ABB RobotStudio station: BARC_MRS_STEP_OPCUA_REV2.rspag

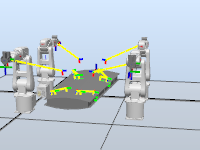
--- station ---
Station BARC_MRS_STEP_OPCUA (saved by RobotStudio 20.1.9014.1)
Controller Rob4, task T_ROB1: task frame (RAPID world) sits at (1193.8, -736.6, 0) mm, rotated rx 0 ry 0 rz -90 deg in the station
Controller Rob3, task T_ROB1: task frame (RAPID world) sits at (0, -736.6, 0) mm, rotated rx 0 ry 0 rz -90 deg in the station
Controller Rob2, task T_ROB1: task frame (RAPID world) sits at (1193.8, 0, 0) mm, rotated rx 0 ry 0 rz 90 deg in the station
Controller Rob1, task T_ROB1: task frame (RAPID world) sits at (0, 0, 0) mm, rotated rx 0 ry 0 rz 90 deg in the station
Controller Rob1
  mechanical unit ROB_1: Rob1, 6 joints, base frame (0, 0, 0) mm
Controller Rob2
  mechanical unit ROB_1: Rob2, 6 joints, base frame (0, 0, 0) mm
Controller Rob3
  mechanical unit ROB_1: Rob3, 6 joints, base frame (0, 0, 0) mm
Controller Rob4
  mechanical unit ROB_1: Rob4, 6 joints, base frame (0, 0, 0) mm
Layout (positions relative to the parent item):
  - Rob1 [mechanism, from Robots\IRB120_3_58_G_01.rslib] at (0, 0, 0) mm, rotated rx 0 ry 0 rz 90 deg; joint values [0, 0, 0, 0, 0, 0] (rad or m)
  - Rob2 [mechanism, from Robots\IRB120_3_58_G_01.rslib] at (1193.8, 0, 0) mm, rotated rx 0 ry 0 rz 90 deg; joint values [0, 0, 0, 0, 0, 0] (rad or m)
  - Rob3 [mechanism, from Robots\IRB120_3_58_G_01.rslib] at (0, -736.6, 0) mm, rotated rx 0 ry 0 rz -90 deg; joint values [0, 0, 0, 0, 0, 0] (rad or m)
  - Rob4 [mechanism, from Robots\IRB120_3_58_G_01.rslib] at (1193.8, -736.6, 0) mm, rotated rx 0 ry 0 rz -90 deg; joint values [0, 0, 0, 0, 0, 0] (rad or m)
  - MyTool [mechanism, from Training Objects\myTool.rslib] at (0, 374, 630) mm, rotated rx 0 ry 90 rz 90 deg
  - MyTool_2 [mechanism, from Training Objects\myTool.rslib] at (1193.8, 374, 630) mm, rotated rx 0 ry 90 rz 90 deg
  - MyTool_3 [mechanism, from Training Objects\myTool.rslib] at (0, -1110.6, 630) mm, rotated rx 0 ry 90 rz -90 deg
  - MyTool_4 [mechanism, from Training Objects\myTool.rslib] at (1193.8, -1110.6, 630) mm, rotated rx 0 ry 90 rz -90 deg
  - ScaledWing_Simple_Corrected [part] at (871.22, 154, 150.3) mm, rotated rx 90 ry 0 rz -90 deg
  - onepiece [part] at (287.65, 225, -913.8) mm, rotated rx 89 ry 0 rz 0 deg
  - PendEff [mechanism, from Libraries\PendEff.rslib] at (0, 374, 630) mm, rotated rx 0 ry 90 rz 90 deg
  - PendEff_2 [mechanism, from Libraries\PendEff.rslib] at (1193.8, 374, 630) mm, rotated rx 0 ry 90 rz 90 deg
  - PendEff_3 [mechanism, from Libraries\PendEff.rslib] at (0, -1110.6, 630) mm, rotated rx 0 ry 90 rz -90 deg
  - PendEff_4 [mechanism, from Libraries\PendEff.rslib] at (1193.8, -1110.6, 630) mm, rotated rx 0 ry 90 rz -90 deg
  - wing_with_holes_2 [part] at (596.5, 225, -913.8) mm, rotated rx 89 ry 0 rz 0 deg
  - Part_1 [part]
  - Part_2 [part]
  - Part_3 [part]
  - Part_4 [part]
  - Part_5 [part]
  - Part_6 [part]
  - Part_7 [part]
  - Part_8 [part]
  - partwithpoints [part, from Libraries\partwithpoints.rslib]
  - SmartComponent_1 [smart component]
Attachment: MyTool is attached to Rob1 / Link6
Attachment: MyTool_2 is attached to Rob2 / Link6
Attachment: MyTool_3 is attached to Rob3 / Link6
Attachment: MyTool_4 is attached to Rob4 / Link6
Attachment: PendEff is attached to Rob1 / Link6
Attachment: PendEff_2 is attached to Rob2 / Link6
Attachment: PendEff_3 is attached to Rob3 / Link6
Attachment: PendEff_4 is attached to Rob4 / Link6
Targets, tools, work objects and paths stored in the station and not in the controller backup, written as RAPID:
! task T_ROB1
MODULE KegleyMod
  PERS speeddata ExternalFedSpeedData:=[100,100,500,500];
  PERS zonedata ExternalFedZoneData:=[True,0,0,0,0,0,0];
ENDMODULE

! task T_ROB1
MODULE StanModule
  PROC STEPpath()
    MoveL current_robtarget,v1000,z100,PendEff_point\WObj:=A;
    SetDO doIsComplete,1;
  ENDPROC
  PROC WorkingStep()
    SetDO doIsComplete,0;
    MoveL current_robtarget,v1000,z100,PendEff_point\WObj:=A;
    SetDO doIsComplete,1;
  ENDPROC
ENDMODULE

! task T_ROB1
MODULE Targets
  CONST robtarget Drilling0:=[[255.049346094,-251.794133959,27.074601391],[0.009317717,-0.000993284,-0.994322357,-0.105996434],[0,0,0,0],[9E+09,9E+09,9E+09,9E+09,9E+09,9E+09]];
  CONST robtarget Drilling1:=[[254.118737842,-241.085099842,-22.575076921],[0.009317717,-0.000993284,-0.994322357,-0.105996434],[0,0,0,0],[9E+09,9E+09,9E+09,9E+09,9E+09,9E+09]];
  CONST robtarget Drilling2:=[[254.118737842,-241.085099842,-22.575076921],[0.009317717,-0.000993284,-0.994322357,-0.105996434],[0,0,0,0],[9E+09,9E+09,9E+09,9E+09,9E+09,9E+09]];
  CONST robtarget Drilling3:=[[253.537107684,-234.391953519,-53.606125867],[0.009317717,-0.000993284,-0.994322357,-0.105996434],[0,0,0,0],[9E+09,9E+09,9E+09,9E+09,9E+09,9E+09]];
  CONST robtarget Drilling4:=[[253.537107684,-234.391953519,-53.606125867],[0.009317717,-0.000993284,-0.994322357,-0.105996434],[0,0,0,0],[9E+09,9E+09,9E+09,9E+09,9E+09,9E+09]];
  CONST robtarget Drilling5:=[[254.118737842,-241.085099842,-22.575076921],[0.009317717,-0.000993284,-0.994322357,-0.105996434],[0,0,0,0],[9E+09,9E+09,9E+09,9E+09,9E+09,9E+09]];
  CONST robtarget Drilling6:=[[255.049346094,-251.794133959,27.074601391],[0.009317717,-0.000993284,-0.994322357,-0.105996434],[0,0,0,0],[9E+09,9E+09,9E+09,9E+09,9E+09,9E+09]];
  CONST robtarget Drilling7:=[[593.951420596,-86.046366407,46.267647759],[0.006736064,-0.000262673,-0.999217855,-0.038964529],[0,0,0,0],[9E+09,9E+09,9E+09,9E+09,9E+09,9E+09]];
  CONST robtarget Drilling8:=[[593.268611665,-82.090486811,-4.373489556],[0.006736064,-0.000262673,-0.999217855,-0.038964529],[0,0,0,0],[9E+09,9E+09,9E+09,9E+09,9E+09,9E+09]];
  CONST robtarget Drilling9:=[[593.268611665,-82.090486811,-4.373489556],[0.006736064,-0.000262673,-0.999217855,-0.038964529],[0,0,0,0],[9E+09,9E+09,9E+09,9E+09,9E+09,9E+09]];
  CONST robtarget Drilling10:=[[592.841856083,-79.618062064,-36.024200378],[0.006736064,-0.000262673,-0.999217855,-0.038964529],[0,0,0,0],[9E+09,9E+09,9E+09,9E+09,9E+09,9E+09]];
  CONST robtarget Drilling11:=[[592.841856083,-79.618062064,-36.024200378],[0.006736064,-0.000262673,-0.999217855,-0.038964529],[0,0,0,0],[9E+09,9E+09,9E+09,9E+09,9E+09,9E+09]];
  CONST robtarget Drilling12:=[[593.268611665,-82.090486811,-4.373489556],[0.006736064,-0.000262673,-0.999217855,-0.038964529],[0,0,0,0],[9E+09,9E+09,9E+09,9E+09,9E+09,9E+09]];
  CONST robtarget Drilling13:=[[593.951420596,-86.046366407,46.267647759],[0.006736064,-0.000262673,-0.999217855,-0.038964529],[0,0,0,0],[9E+09,9E+09,9E+09,9E+09,9E+09,9E+09]];
  CONST robtarget Drilling14:=[[594.013579836,-136.119059315,41.206016458],[0.007335405,-0.000453474,-0.998067656,-0.061700413],[0,0,0,0],[9E+09,9E+09,9E+09,9E+09,9E+09,9E+09]];
  CONST robtarget Drilling15:=[[593.272585499,-129.86207284,-9.201731435],[0.007335405,-0.000453474,-0.998067656,-0.061700413],[0,0,0,0],[9E+09,9E+09,9E+09,9E+09,9E+09,9E+09]];
  CONST robtarget Drilling16:=[[593.272585499,-129.86207284,-9.201731435],[0.007335405,-0.000453474,-0.998067656,-0.061700413],[0,0,0,0],[9E+09,9E+09,9E+09,9E+09,9E+09,9E+09]];
  CONST robtarget Drilling17:=[[592.809464038,-125.951456293,-40.706573868],[0.007335405,-0.000453474,-0.998067656,-0.061700413],[0,0,0,0],[9E+09,9E+09,9E+09,9E+09,9E+09,9E+09]];
  CONST robtarget Drilling18:=[[592.809464038,-125.951456293,-40.706573868],[0.007335405,-0.000453474,-0.998067656,-0.061700413],[0,0,0,0],[9E+09,9E+09,9E+09,9E+09,9E+09,9E+09]];
  CONST robtarget Drilling19:=[[593.272585499,-129.86207284,-9.201731435],[0.007335405,-0.000453474,-0.998067656,-0.061700413],[0,0,0,0],[9E+09,9E+09,9E+09,9E+09,9E+09,9E+09]];
  CONST robtarget Drilling20:=[[594.013579836,-136.119059315,41.206016458],[0.007335405,-0.000453474,-0.998067656,-0.061700413],[0,0,0,0],[9E+09,9E+09,9E+09,9E+09,9E+09,9E+09]];
  PROC dummy()
    MoveL Drilling0,v0,z10,DrillTool\WObj:=A;
    MoveL Drilling1,v1,z10,DrillTool\WObj:=A;
    MoveL Drilling2,v2,z10,DrillTool\WObj:=A;
    MoveL Drilling3,v3,z10,DrillTool\WObj:=A;
    MoveL Drilling4,v4,z10,DrillTool\WObj:=A;
    MoveL Drilling5,v5,z10,DrillTool\WObj:=A;
    MoveL Drilling6,v6,z10,DrillTool\WObj:=A;
    MoveL Drilling7,v7,z10,DrillTool\WObj:=A;
    MoveL Drilling8,v8,z10,DrillTool\WObj:=A;
    MoveL Drilling9,v9,z10,DrillTool\WObj:=A;
    MoveL Drilling10,v10,z10,DrillTool\WObj:=A;
    MoveL Drilling11,v11,z10,DrillTool\WObj:=A;
    MoveL Drilling12,v12,z10,DrillTool\WObj:=A;
    MoveL Drilling13,v13,z10,DrillTool\WObj:=A;
    MoveL Drilling14,v14,z10,DrillTool\WObj:=A;
    MoveL Drilling15,v15,z10,DrillTool\WObj:=A;
    MoveL Drilling16,v16,z10,DrillTool\WObj:=A;
    MoveL Drilling17,v17,z10,DrillTool\WObj:=A;
    MoveL Drilling18,v18,z10,DrillTool\WObj:=A;
    MoveL Drilling19,v19,z10,DrillTool\WObj:=A;
    MoveL Drilling20,v20,z10,DrillTool\WObj:=A;
  ENDPROC
ENDMODULE

! task T_ROB1
MODULE KegleyMod
  PERS speeddata ExternalFedSpeedData:=[100,100,500,500];
  PERS zonedata ExternalFedZoneData:=[True,0,0,0,0,0,0];
ENDMODULE

! task T_ROB1
MODULE KyleModule
  PROC WorkingStep()
    SetDO doIsComplete,0;
    MoveL current_robtarget,v1000,z100,PendEff_point\WObj:=A;
    SetDO doIsComplete,1;
  ENDPROC
ENDMODULE

! task T_ROB1
MODULE Targets
  CONST robtarget Drilling0:=[[241.166080887,78.477337456,51.523766918],[0.006620989,0.000217104,-0.999440903,0.032771904],[0,0,0,0],[9E+09,9E+09,9E+09,9E+09,9E+09,9E+09]];
  CONST robtarget Drilling1:=[[240.494487367,75.149427584,0.837338971],[0.006620989,0.000217104,-0.999440903,0.032771904],[0,0,0,0],[9E+09,9E+09,9E+09,9E+09,9E+09,9E+09]];
  CONST robtarget Drilling2:=[[240.494487367,75.149427584,0.837338971],[0.006620989,0.000217104,-0.999440903,0.032771904],[0,0,0,0],[9E+09,9E+09,9E+09,9E+09,9E+09,9E+09]];
  CONST robtarget Drilling3:=[[240.074741417,73.069483914,-30.841678495],[0.006620989,0.000217104,-0.999440903,0.032771904],[0,0,0,0],[9E+09,9E+09,9E+09,9E+09,9E+09,9E+09]];
  CONST robtarget Drilling4:=[[240.074741417,73.069483914,-30.841678495],[0.006620989,0.000217104,-0.999440903,0.032771904],[0,0,0,0],[9E+09,9E+09,9E+09,9E+09,9E+09,9E+09]];
  CONST robtarget Drilling5:=[[240.494487367,75.149427584,0.837338971],[0.006620989,0.000217104,-0.999440903,0.032771904],[0,0,0,0],[9E+09,9E+09,9E+09,9E+09,9E+09,9E+09]];
  CONST robtarget Drilling6:=[[241.166080887,78.477337456,51.523766918],[0.006620989,0.000217104,-0.999440903,0.032771904],[0,0,0,0],[9E+09,9E+09,9E+09,9E+09,9E+09,9E+09]];
  CONST robtarget Drilling7:=[[590.794286308,244.057268889,22.395212352],[0.009603198,0.001072712,-0.993772536,0.111007991],[0,0,0,0],[9E+09,9E+09,9E+09,9E+09,9E+09,9E+09]];
  CONST robtarget Drilling8:=[[589.836775887,232.848046285,-27.143424109],[0.009603198,0.001072712,-0.993772536,0.111007991],[0,0,0,0],[9E+09,9E+09,9E+09,9E+09,9E+09,9E+09]];
  CONST robtarget Drilling9:=[[589.836775887,232.848046285,-27.143424109],[0.009603198,0.001072712,-0.993772536,0.111007991],[0,0,0,0],[9E+09,9E+09,9E+09,9E+09,9E+09,9E+09]];
  CONST robtarget Drilling10:=[[589.238331874,225.842282157,-58.105071897],[0.009603198,0.001072712,-0.993772536,0.111007991],[0,0,0,0],[9E+09,9E+09,9E+09,9E+09,9E+09,9E+09]];
  CONST robtarget Drilling11:=[[589.238331874,225.842282157,-58.105071897],[0.009603198,0.001072712,-0.993772536,0.111007991],[0,0,0,0],[9E+09,9E+09,9E+09,9E+09,9E+09,9E+09]];
  CONST robtarget Drilling12:=[[589.836775887,232.848046285,-27.143424109],[0.009603198,0.001072712,-0.993772536,0.111007991],[0,0,0,0],[9E+09,9E+09,9E+09,9E+09,9E+09,9E+09]];
  CONST robtarget Drilling13:=[[590.794286308,244.057268889,22.395212352],[0.009603198,0.001072712,-0.993772536,0.111007991],[0,0,0,0],[9E+09,9E+09,9E+09,9E+09,9E+09,9E+09]];
  CONST robtarget Drilling14:=[[586.927237976,164.129102175,37.475265565],[0.00778853,0.000580627,-0.997202343,0.074340359],[0,0,0,0],[9E+09,9E+09,9E+09,9E+09,9E+09,9E+09]];
  CONST robtarget Drilling15:=[[586.142522602,156.59679287,-12.757079974],[0.00778853,0.000580627,-0.997202343,0.074340359],[0,0,0,0],[9E+09,9E+09,9E+09,9E+09,9E+09,9E+09]];
  CONST robtarget Drilling16:=[[586.142522602,156.59679287,-12.757079974],[0.00778853,0.000580627,-0.997202343,0.074340359],[0,0,0,0],[9E+09,9E+09,9E+09,9E+09,9E+09,9E+09]];
  CONST robtarget Drilling17:=[[585.652075493,151.889099555,-44.152295936],[0.00778853,0.000580627,-0.997202343,0.074340359],[0,0,0,0],[9E+09,9E+09,9E+09,9E+09,9E+09,9E+09]];
  CONST robtarget Drilling18:=[[585.652075493,151.889099555,-44.152295936],[0.00778853,0.000580627,-0.997202343,0.074340359],[0,0,0,0],[9E+09,9E+09,9E+09,9E+09,9E+09,9E+09]];
  CONST robtarget Drilling19:=[[586.142522602,156.59679287,-12.757079974],[0.00778853,0.000580627,-0.997202343,0.074340359],[0,0,0,0],[9E+09,9E+09,9E+09,9E+09,9E+09,9E+09]];
  CONST robtarget Drilling20:=[[586.927237976,164.129102175,37.475265565],[0.00778853,0.000580627,-0.997202343,0.074340359],[0,0,0,0],[9E+09,9E+09,9E+09,9E+09,9E+09,9E+09]];
  PROC dummy()
    MoveL Drilling0,v0,z10,DrillTool\WObj:=A;
    MoveL Drilling1,v1,z10,DrillTool\WObj:=A;
    MoveL Drilling2,v2,z10,DrillTool\WObj:=A;
    MoveL Drilling3,v3,z10,DrillTool\WObj:=A;
    MoveL Drilling4,v4,z10,DrillTool\WObj:=A;
    MoveL Drilling5,v5,z10,DrillTool\WObj:=A;
    MoveL Drilling6,v6,z10,DrillTool\WObj:=A;
    MoveL Drilling7,v7,z10,DrillTool\WObj:=A;
    MoveL Drilling8,v8,z10,DrillTool\WObj:=A;
    MoveL Drilling9,v9,z10,DrillTool\WObj:=A;
    MoveL Drilling10,v10,z10,DrillTool\WObj:=A;
    MoveL Drilling11,v11,z10,DrillTool\WObj:=A;
    MoveL Drilling12,v12,z10,DrillTool\WObj:=A;
    MoveL Drilling13,v13,z10,DrillTool\WObj:=A;
    MoveL Drilling14,v14,z10,DrillTool\WObj:=A;
    MoveL Drilling15,v15,z10,DrillTool\WObj:=A;
    MoveL Drilling16,v16,z10,DrillTool\WObj:=A;
    MoveL Drilling17,v17,z10,DrillTool\WObj:=A;
    MoveL Drilling18,v18,z10,DrillTool\WObj:=A;
    MoveL Drilling19,v19,z10,DrillTool\WObj:=A;
    MoveL Drilling20,v20,z10,DrillTool\WObj:=A;
  ENDPROC
ENDMODULE

! task T_ROB1
MODULE KegleyMod
  PERS speeddata ExternalFedSpeedData:=[100,100,500,500];
  PERS zonedata ExternalFedZoneData:=[True,0,0,0,0,0,0];
ENDMODULE

! task T_ROB1
MODULE CartmanWorkingPlan
  PROC WorkingStep()
    SetDO doIsComplete,0;
    MoveL current_robtarget,v1000,z100,PendEff_point\WObj:=A;
    SetDO doIsComplete,1;
  ENDPROC
ENDMODULE

! task T_ROB1
MODULE Targets
  CONST robtarget Drilling0:=[[1189.808543498,-65.923675679,39.773088683],[0.006653359,-0.000231419,-0.9993735,-0.034760413],[0,0,0,0],[9E+09,9E+09,9E+09,9E+09,9E+09,9E+09]];
  CONST robtarget Drilling1:=[[1189.133802971,-62.394073863,-10.899651881],[0.006653359,-0.000231419,-0.9993735,-0.034760413],[0,0,0,0],[9E+09,9E+09,9E+09,9E+09,9E+09,9E+09]];
  CONST robtarget Drilling2:=[[1189.133802971,-62.394073863,-10.899651881],[0.006653359,-0.000231419,-0.9993735,-0.034760413],[0,0,0,0],[9E+09,9E+09,9E+09,9E+09,9E+09,9E+09]];
  CONST robtarget Drilling3:=[[1188.712090141,-60.188072728,-42.570114734],[0.006653359,-0.000231419,-0.9993735,-0.034760413],[0,0,0,0],[9E+09,9E+09,9E+09,9E+09,9E+09,9E+09]];
  CONST robtarget Drilling4:=[[1188.712090141,-60.188072728,-42.570114734],[0.006653359,-0.000231419,-0.9993735,-0.034760413],[0,0,0,0],[9E+09,9E+09,9E+09,9E+09,9E+09,9E+09]];
  CONST robtarget Drilling5:=[[1189.133802971,-62.394073863,-10.899651881],[0.006653359,-0.000231419,-0.9993735,-0.034760413],[0,0,0,0],[9E+09,9E+09,9E+09,9E+09,9E+09,9E+09]];
  CONST robtarget Drilling6:=[[1189.808543498,-65.923675679,39.773088683],[0.006653359,-0.000231419,-0.9993735,-0.034760413],[0,0,0,0],[9E+09,9E+09,9E+09,9E+09,9E+09,9E+09]];
  CONST robtarget Drilling7:=[[1275.333810152,-199.568058709,19.231409467],[0.009422515,-0.001026722,-0.994071031,-0.10831873],[0,0,0,0],[9E+09,9E+09,9E+09,9E+09,9E+09,9E+09]];
  CONST robtarget Drilling8:=[[1274.39345782,-188.627142215,-30.367502656],[0.009422515,-0.001026722,-0.994071031,-0.10831873],[0,0,0,0],[9E+09,9E+09,9E+09,9E+09,9E+09,9E+09]];
  CONST robtarget Drilling9:=[[1274.39345782,-188.627142215,-30.367502656],[0.009422515,-0.001026722,-0.994071031,-0.10831873],[0,0,0,0],[9E+09,9E+09,9E+09,9E+09,9E+09,9E+09]];
  CONST robtarget Drilling10:=[[1273.805737613,-181.789069407,-61.366822732],[0.009422515,-0.001026722,-0.994071031,-0.10831873],[0,0,0,0],[9E+09,9E+09,9E+09,9E+09,9E+09,9E+09]];
  CONST robtarget Drilling11:=[[1273.805737613,-181.789069407,-61.366822732],[0.009422515,-0.001026722,-0.994071031,-0.10831873],[0,0,0,0],[9E+09,9E+09,9E+09,9E+09,9E+09,9E+09]];
  CONST robtarget Drilling12:=[[1274.39345782,-188.627142215,-30.367502656],[0.009422515,-0.001026722,-0.994071031,-0.10831873],[0,0,0,0],[9E+09,9E+09,9E+09,9E+09,9E+09,9E+09]];
  CONST robtarget Drilling13:=[[1275.333810152,-199.568058709,19.231409467],[0.009422515,-0.001026722,-0.994071031,-0.10831873],[0,0,0,0],[9E+09,9E+09,9E+09,9E+09,9E+09,9E+09]];
  CONST robtarget Drilling14:=[[1277.649426378,-158.123953639,27.348886106],[0.008256342,-0.000710159,-0.996287003,-0.085694437],[0,0,0,0],[9E+09,9E+09,9E+09,9E+09,9E+09,9E+09]];
  CONST robtarget Drilling15:=[[1276.819879727,-149.449130571,-22.698084803],[0.008256342,-0.000710159,-0.996287003,-0.085694437],[0,0,0,0],[9E+09,9E+09,9E+09,9E+09,9E+09,9E+09]];
  CONST robtarget Drilling16:=[[1276.819879727,-149.449130571,-22.698084803],[0.008256342,-0.000710159,-0.996287003,-0.085694437],[0,0,0,0],[9E+09,9E+09,9E+09,9E+09,9E+09,9E+09]];
  CONST robtarget Drilling17:=[[1276.30141307,-144.027366153,-53.97744162],[0.008256342,-0.000710159,-0.996287003,-0.085694437],[0,0,0,0],[9E+09,9E+09,9E+09,9E+09,9E+09,9E+09]];
  CONST robtarget Drilling18:=[[1276.30141307,-144.027366153,-53.97744162],[0.008256342,-0.000710159,-0.996287003,-0.085694437],[0,0,0,0],[9E+09,9E+09,9E+09,9E+09,9E+09,9E+09]];
  CONST robtarget Drilling19:=[[1276.819879727,-149.449130571,-22.698084803],[0.008256342,-0.000710159,-0.996287003,-0.085694437],[0,0,0,0],[9E+09,9E+09,9E+09,9E+09,9E+09,9E+09]];
  CONST robtarget Drilling20:=[[1277.649426378,-158.123953639,27.348886106],[0.008256342,-0.000710159,-0.996287003,-0.085694437],[0,0,0,0],[9E+09,9E+09,9E+09,9E+09,9E+09,9E+09]];
  PROC dummy()
    MoveL Drilling0,v0,z10,DrillTool\WObj:=A;
    MoveL Drilling1,v1,z10,DrillTool\WObj:=A;
    MoveL Drilling2,v2,z10,DrillTool\WObj:=A;
    MoveL Drilling3,v3,z10,DrillTool\WObj:=A;
    MoveL Drilling4,v4,z10,DrillTool\WObj:=A;
    MoveL Drilling5,v5,z10,DrillTool\WObj:=A;
    MoveL Drilling6,v6,z10,DrillTool\WObj:=A;
    MoveL Drilling7,v7,z10,DrillTool\WObj:=A;
    MoveL Drilling8,v8,z10,DrillTool\WObj:=A;
    MoveL Drilling9,v9,z10,DrillTool\WObj:=A;
    MoveL Drilling10,v10,z10,DrillTool\WObj:=A;
    MoveL Drilling11,v11,z10,DrillTool\WObj:=A;
    MoveL Drilling12,v12,z10,DrillTool\WObj:=A;
    MoveL Drilling13,v13,z10,DrillTool\WObj:=A;
    MoveL Drilling14,v14,z10,DrillTool\WObj:=A;
    MoveL Drilling15,v15,z10,DrillTool\WObj:=A;
    MoveL Drilling16,v16,z10,DrillTool\WObj:=A;
    MoveL Drilling17,v17,z10,DrillTool\WObj:=A;
    MoveL Drilling18,v18,z10,DrillTool\WObj:=A;
    MoveL Drilling19,v19,z10,DrillTool\WObj:=A;
    MoveL Drilling20,v20,z10,DrillTool\WObj:=A;
  ENDPROC
ENDMODULE

! task T_ROB1
MODULE KegleyMod
  PERS speeddata ExternalFedSpeedData:=[100,100,500,500];
  PERS zonedata ExternalFedZoneData:=[True,0,0,0,0,0,0];
ENDMODULE

! task T_ROB1
MODULE Targets
  CONST robtarget Drilling0:=[[1191.894155606,213.973804454,17.582383099],[0.009735859,0.001112565,-0.993486175,0.11353059],[0,0,0,0],[9E+09,9E+09,9E+09,9E+09,9E+09,9E+09]];
  CONST robtarget Drilling1:=[[1190.924268649,202.513131068,-31.898444348],[0.009735859,0.001112565,-0.993486175,0.11353059],[0,0,0,0],[9E+09,9E+09,9E+09,9E+09,9E+09,9E+09]];
  CONST robtarget Drilling2:=[[1190.924268649,202.513131068,-31.898444348],[0.009735859,0.001112565,-0.993486175,0.11353059],[0,0,0,0],[9E+09,9E+09,9E+09,9E+09,9E+09,9E+09]];
  CONST robtarget Drilling3:=[[1190.318089301,195.350210202,-62.823961503],[0.009735859,0.001112565,-0.993486175,0.11353059],[0,0,0,0],[9E+09,9E+09,9E+09,9E+09,9E+09,9E+09]];
  CONST robtarget Drilling4:=[[1190.318089301,195.350210202,-62.823961503],[0.009735859,0.001112565,-0.993486175,0.11353059],[0,0,0,0],[9E+09,9E+09,9E+09,9E+09,9E+09,9E+09]];
  CONST robtarget Drilling5:=[[1190.924268649,202.513131068,-31.898444348],[0.009735859,0.001112565,-0.993486175,0.11353059],[0,0,0,0],[9E+09,9E+09,9E+09,9E+09,9E+09,9E+09]];
  CONST robtarget Drilling6:=[[1191.894155606,213.973804454,17.582383099],[0.009735859,0.001112565,-0.993486175,0.11353059],[0,0,0,0],[9E+09,9E+09,9E+09,9E+09,9E+09,9E+09]];
  CONST robtarget Drilling7:=[[1279.805555756,62.025883801,38.843455502],[0.006631324,0.000222501,-0.999415571,0.033533444],[0,0,0,0],[9E+09,9E+09,9E+09,9E+09,9E+09,9E+09]];
  CONST robtarget Drilling8:=[[1279.132965076,58.620727156,-11.837828321],[0.006631324,0.000222501,-0.999415571,0.033533444],[0,0,0,0],[9E+09,9E+09,9E+09,9E+09,9E+09,9E+09]];
  CONST robtarget Drilling9:=[[1279.132965076,58.620727156,-11.837828321],[0.006631324,0.000222501,-0.999415571,0.033533444],[0,0,0,0],[9E+09,9E+09,9E+09,9E+09,9E+09,9E+09]];
  CONST robtarget Drilling10:=[[1278.712595901,56.492504252,-43.513630711],[0.006631324,0.000222501,-0.999415571,0.033533444],[0,0,0,0],[9E+09,9E+09,9E+09,9E+09,9E+09,9E+09]];
  CONST robtarget Drilling11:=[[1278.712595901,56.492504252,-43.513630711],[0.006631324,0.000222501,-0.999415571,0.033533444],[0,0,0,0],[9E+09,9E+09,9E+09,9E+09,9E+09,9E+09]];
  CONST robtarget Drilling12:=[[1279.132965076,58.620727156,-11.837828321],[0.006631324,0.000222501,-0.999415571,0.033533444],[0,0,0,0],[9E+09,9E+09,9E+09,9E+09,9E+09,9E+09]];
  CONST robtarget Drilling13:=[[1279.805555756,62.025883801,38.843455502],[0.006631324,0.000222501,-0.999415571,0.033533444],[0,0,0,0],[9E+09,9E+09,9E+09,9E+09,9E+09,9E+09]];
  CONST robtarget Drilling14:=[[1280.462702991,102.383093395,35.233257482],[0.007136454,0.000396072,-0.998437928,0.055413159],[0,0,0,0],[9E+09,9E+09,9E+09,9E+09,9E+09,9E+09]];
  CONST robtarget Drilling15:=[[1279.741001712,96.761623708,-15.249593327],[0.007136454,0.000396072,-0.998437928,0.055413159],[0,0,0,0],[9E+09,9E+09,9E+09,9E+09,9E+09,9E+09]];
  CONST robtarget Drilling16:=[[1279.741001712,96.761623708,-15.249593327],[0.007136454,0.000396072,-0.998437928,0.055413159],[0,0,0,0],[9E+09,9E+09,9E+09,9E+09,9E+09,9E+09]];
  CONST robtarget Drilling17:=[[1279.289938413,93.248205154,-46.801375083],[0.007136454,0.000396072,-0.998437928,0.055413159],[0,0,0,0],[9E+09,9E+09,9E+09,9E+09,9E+09,9E+09]];
  CONST robtarget Drilling18:=[[1279.289938413,93.248205154,-46.801375083],[0.007136454,0.000396072,-0.998437928,0.055413159],[0,0,0,0],[9E+09,9E+09,9E+09,9E+09,9E+09,9E+09]];
  CONST robtarget Drilling19:=[[1279.741001712,96.761623708,-15.249593327],[0.007136454,0.000396072,-0.998437928,0.055413159],[0,0,0,0],[9E+09,9E+09,9E+09,9E+09,9E+09,9E+09]];
  CONST robtarget Drilling20:=[[1280.462702991,102.383093395,35.233257482],[0.007136454,0.000396072,-0.998437928,0.055413159],[0,0,0,0],[9E+09,9E+09,9E+09,9E+09,9E+09,9E+09]];
  PROC dummy()
    MoveL Drilling0,v0,z10,DrillTool\WObj:=A;
    MoveL Drilling1,v1,z10,DrillTool\WObj:=A;
    MoveL Drilling2,v2,z10,DrillTool\WObj:=A;
    MoveL Drilling3,v3,z10,DrillTool\WObj:=A;
    MoveL Drilling4,v4,z10,DrillTool\WObj:=A;
    MoveL Drilling5,v5,z10,DrillTool\WObj:=A;
    MoveL Drilling6,v6,z10,DrillTool\WObj:=A;
    MoveL Drilling7,v7,z10,DrillTool\WObj:=A;
    MoveL Drilling8,v8,z10,DrillTool\WObj:=A;
    MoveL Drilling9,v9,z10,DrillTool\WObj:=A;
    MoveL Drilling10,v10,z10,DrillTool\WObj:=A;
    MoveL Drilling11,v11,z10,DrillTool\WObj:=A;
    MoveL Drilling12,v12,z10,DrillTool\WObj:=A;
    MoveL Drilling13,v13,z10,DrillTool\WObj:=A;
    MoveL Drilling14,v14,z10,DrillTool\WObj:=A;
    MoveL Drilling15,v15,z10,DrillTool\WObj:=A;
    MoveL Drilling16,v16,z10,DrillTool\WObj:=A;
    MoveL Drilling17,v17,z10,DrillTool\WObj:=A;
    MoveL Drilling18,v18,z10,DrillTool\WObj:=A;
    MoveL Drilling19,v19,z10,DrillTool\WObj:=A;
    MoveL Drilling20,v20,z10,DrillTool\WObj:=A;
  ENDPROC
ENDMODULE

! task T_ROB1
MODULE KennyWorkingPlan
  PROC WorkingStep()
    SetDO doIsComplete,0;
    MoveL current_robtarget,v1000,z100,PendEff_point\WObj:=A;
    SetDO doIsComplete,1;
  ENDPROC
ENDMODULE


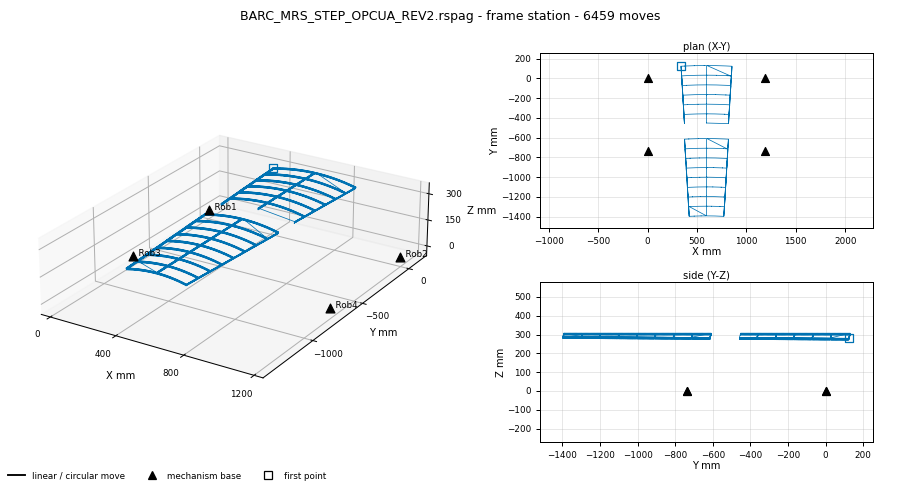
[picture p0: tool path of BARC_MRS_STEP_OPCUA_REV2.rspag in frame station, 6459 of 6483 moves have a stored position in this frame; points joined in program order, loops and branches not executed]
--- Backups/Rob1/RAPID/TASK1/PROGMOD/StanTargets.mod ---
MODULE StanTargets

	!Workplan Variables
	CONST string workplanName := "Stan";
	CONST string workplanUUID := "45926d04-bc6f-4ba0-8e9a-a41acb7af52a";

	!Workingsteps
	CONST string WorkPlan{20,6} := [
		["1","7", "Drilling.2", "b062b09d-c75e-4509-b058-f533fc3121cb", "Hole.101", "7ba2387a-5122-471d-9e62-f4dd978dd916"],
		["8","14", "Drilling.19", "bc6d7e2e-2011-44a2-96ea-1bdf43305bb2", "Hole.2", "a5a2d4b3-bce9-4376-9a01-39ac46aa03b7"],
		["15","21", "Drilling.20", "1d99434e-626c-49cd-aa28-89c40de30f06", "Hole.105", "77f1627f-4d66-488f-b970-3b2b6af52deb"],
		["22","28", "Drilling.3", "45a28ad3-0738-4ba8-bc95-27ca5d3c2a9d", "Hole.102", "83a55789-a548-457f-bc7a-c5f73e279b59"],
		["29","35", "Drilling.1", "9e701cf1-a52e-421d-a5d1-a7fe2dbaa640", "Hole.100", "ec9e4cb9-16a2-432e-8136-2d658a3c3d31"],
		["36","42", "Drilling.18", "90b44a9d-16c4-4a88-bf09-b7f65aff8308", "Hole.106", "8309f7bd-9ba6-4400-9e0b-e392acc79543"],
		["43","49", "Drilling.4", "301b61b0-be88-4471-af20-9d54f270abc0", "Hole.103", "543c12c8-ac8b-46e2-b23c-ed2f3937359b"],
		["50","56", "Drilling.17", "4a6a49de-cb15-4803-8bb7-097c767e5d1a", "Hole.107", "bc5d4dfc-6aa2-4544-8bb1-6cd32004e75e"],
		["57","63", "Drilling.21", "d6a29b26-5ed6-4fc9-a609-95bc5c10512a", "Hole.109", "c5793a88-d117-412a-8380-89480e2aa149"],
		["64","70", "Drilling.22", "32b13ef1-a017-413c-926d-f3ce9280a815", "Hole.110", "f43400ad-c29f-4157-ba87-1fd86718dbb4"],
		["71","77", "Drilling.23", "961958d8-0134-4891-910a-03c3b0fd50ac", "Hole.111", "4c4ae24f-0e25-46c1-affc-8b190d84e835"],
		["78","84", "Drilling.24", "46b8f9da-afaf-476f-bebf-76b29446400a", "Hole.112", "58a054b0-4018-4bcc-8be0-6224a9ae077a"],
		["85","91", "Drilling.37", "a26de890-fc0a-49b5-bfdf-50d0ba577d7f", "Hole.117", "fd2c949e-3c41-489a-8a46-dd0d10567b1b"],
		["92","98", "Drilling.38", "57e6c193-12b5-426e-af89-bc1afa04e779", "Hole.116", "13521d27-8989-4ee6-aa90-747ab0996569"],
		["99","105", "Drilling.39", "43fec44c-5451-4481-a3ed-f2154e5b5857", "Hole.115", "b8ea09e7-7ee5-4781-9867-97bdf0c7c8c2"],
		["106","112", "Drilling.40", "b2407ed9-3760-41ef-9af3-e4b017b94bad", "Hole.114", "6fd1afc0-306a-4e0e-985a-70eb87f380a3"],
		["113","119", "Drilling.41", "e4391847-02d9-4746-a9c4-e995e37bf0a5", "Hole.119", "2fe5694b-30b9-4983-885c-0907e4daf0a7"],
		["120","126", "Drilling.42", "9648c8b5-7603-4606-8e84-4fa243c23e6f", "Hole.120", "7e69786d-15ab-4ddf-bc4f-041c788858b9"],
		["127","133", "Drilling.43", "1797812d-a7bf-4001-89eb-f8bf3d30d00a", "Hole.121", "a39c1e68-904f-4878-9c68-b76c3ab1c433"],
		["134","140", "Drilling.44", "c9657693-5bc7-40ba-995c-70b253dd4bce", "Hole.122", "35b9f3e4-dbe9-4a3b-b0cd-96909b64c764"]
		];

	!Positions
	CONST robtarget WorkingstepRobtargets{140} := [
		[[289.186156636195,-206.403560128169,35.3771625636731],[0.00835255338347923,-0.000732758938354189,-0.996138888459216,-0.0873900040940131],[0,0,0,0],[9E+09,9E+09,9E+09,9E+09,9E+09,9E+09]],
		[[288.347319864636,-197.55839601017,-14.6398287952277],[0.00835255338347923,-0.000732758938354189,-0.996138888459216,-0.0873900040940131],[0,0,0,0],[9E+09,9E+09,9E+09,9E+09,9E+09,9E+09]],
		[[288.347319864636,-197.55839601017,-14.6398287952277],[0.00835255338347923,-0.000732758938354189,-0.996138888459216,-0.0873900040940131],[0,0,0,0],[9E+09,9E+09,9E+09,9E+09,9E+09,9E+09]],
		[[287.823046882412,-192.030168436421,-45.9004483945406],[0.00835255338347923,-0.000732758938354189,-0.996138888459216,-0.0873900040940131],[0,0,0,0],[9E+09,9E+09,9E+09,9E+09,9E+09,9E+09]],
		[[287.823046882412,-192.030168436421,-45.9004483945406],[0.00835255338347923,-0.000732758938354189,-0.996138888459216,-0.0873900040940131],[0,0,0,0],[9E+09,9E+09,9E+09,9E+09,9E+09,9E+09]],
		[[288.347319864636,-197.55839601017,-14.6398287952277],[0.00835255338347923,-0.000732758938354189,-0.996138888459216,-0.0873900040940131],[0,0,0,0],[9E+09,9E+09,9E+09,9E+09,9E+09,9E+09]],
		[[289.186156636195,-206.403560128169,35.3771625636731],[0.00835255338347923,-0.000732758938354189,-0.996138888459216,-0.0873900040940131],[0,0,0,0],[9E+09,9E+09,9E+09,9E+09,9E+09,9E+09]],
		[[254.909208192728,-190.980764818536,38.5531834909307],[0.00803255668836741,-0.000646350507138514,-0.996745854533864,-0.0802044994599877],[0,0,0,0],[9E+09,9E+09,9E+09,9E+09,9E+09,9E+09]],
		[[254.101023132797,-182.857977487938,-11.5866924850904],[0.00803255668836741,-0.000646350507138514,-0.996745854533864,-0.0802044994599877],[0,0,0,0],[9E+09,9E+09,9E+09,9E+09,9E+09,9E+09]],
		[[254.101023132797,-182.857977487938,-11.5866924850904],[0.00803255668836741,-0.000646350507138514,-0.996745854533864,-0.0802044994599877],[0,0,0,0],[9E+09,9E+09,9E+09,9E+09,9E+09,9E+09]],
		[[253.595907470339,-177.781235406315,-42.9241149701038],[0.00803255668836741,-0.000646350507138514,-0.996745854533864,-0.0802044994599877],[0,0,0,0],[9E+09,9E+09,9E+09,9E+09,9E+09,9E+09]],
		[[253.595907470339,-177.781235406315,-42.9241149701038],[0.00803255668836741,-0.000646350507138514,-0.996745854533864,-0.0802044994599877],[0,0,0,0],[9E+09,9E+09,9E+09,9E+09,9E+09,9E+09]],
		[[254.101023132797,-182.857977487938,-11.5866924850904],[0.00803255668836741,-0.000646350507138514,-0.996745854533864,-0.0802044994599877],[0,0,0,0],[9E+09,9E+09,9E+09,9E+09,9E+09,9E+09]],
		[[254.909208192728,-190.980764818536,38.5531834909307],[0.00803255668836741,-0.000646350507138514,-0.996745854533864,-0.0802044994599877],[0,0,0,0],[9E+09,9E+09,9E+09,9E+09,9E+09,9E+09]],
		[[255.049346094491,-251.794133959213,27.0746013914174],[0.00931771731230624,-0.000993284320775785,-0.994322356952738,-0.105996433875385],[0,0,0,0],[9E+09,9E+09,9E+09,9E+09,9E+09,9E+09]],
		[[254.118737842067,-241.085099842443,-22.5750769214012],[0.00931771731230624,-0.000993284320775785,-0.994322356952738,-0.105996433875385],[0,0,0,0],[9E+09,9E+09,9E+09,9E+09,9E+09,9E+09]],
		[[254.118737842067,-241.085099842443,-22.5750769214012],[0.00931771731230624,-0.000993284320775785,-0.994322356952738,-0.105996433875385],[0,0,0,0],[9E+09,9E+09,9E+09,9E+09,9E+09,9E+09]],
		[[253.5371076843,-234.391953519461,-53.6061258669128],[0.00931771731230624,-0.000993284320775785,-0.994322356952738,-0.105996433875385],[0,0,0,0],[9E+09,9E+09,9E+09,9E+09,9E+09,9E+09]],
		[[253.5371076843,-234.391953519461,-53.6061258669128],[0.00931771731230624,-0.000993284320775785,-0.994322356952738,-0.105996433875385],[0,0,0,0],[9E+09,9E+09,9E+09,9E+09,9E+09,9E+09]],
		[[254.118737842067,-241.085099842443,-22.5750769214012],[0.00931771731230624,-0.000993284320775785,-0.994322356952738,-0.105996433875385],[0,0,0,0],[9E+09,9E+09,9E+09,9E+09,9E+09,9E+09]],
		[[255.049346094491,-251.794133959213,27.0746013914174],[0.00931771731230624,-0.000993284320775785,-0.994322356952738,-0.105996433875385],[0,0,0,0],[9E+09,9E+09,9E+09,9E+09,9E+09,9E+09]],
		[[288.817292795415,-151.336810998548,43.7919561194079],[0.00741254609803812,-0.000475090293762373,-0.997924837913392,-0.0639597242417948],[0,0,0,0],[9E+09,9E+09,9E+09,9E+09,9E+09,9E+09]],
		[[288.068828229942,-144.851630260459,-6.58683139665437],[0.00741254609803812,-0.000475090293762373,-0.997924837913392,-0.0639597242417948],[0,0,0,0],[9E+09,9E+09,9E+09,9E+09,9E+09,9E+09]],
		[[288.068828229942,-144.851630260459,-6.58683139665437],[0.00741254609803812,-0.000475090293762373,-0.997924837913392,-0.0639597242417948],[0,0,0,0],[9E+09,9E+09,9E+09,9E+09,9E+09,9E+09]],
		[[287.60103787652,-140.798392299153,-38.0735735941933],[0.00741254609803812,-0.000475090293762373,-0.997924837913392,-0.0639597242417948],[0,0,0,0],[9E+09,9E+09,9E+09,9E+09,9E+09,9E+09]],
		[[287.60103787652,-140.798392299153,-38.0735735941933],[0.00741254609803812,-0.000475090293762373,-0.997924837913392,-0.0639597242417948],[0,0,0,0],[9E+09,9E+09,9E+09,9E+09,9E+09,9E+09]],
		[[288.068828229942,-144.851630260459,-6.58683139665437],[0.00741254609803812,-0.000475090293762373,-0.997924837913392,-0.0639597242417948],[0,0,0,0],[9E+09,9E+09,9E+09,9E+09,9E+09,9E+09]],
		[[288.817292795415,-151.336810998548,43.7919561194079],[0.00741254609803812,-0.000475090293762373,-0.997924837913392,-0.0639597242417948],[0,0,0,0],[9E+09,9E+09,9E+09,9E+09,9E+09,9E+09]],
		[[293.28700751171,-244.361649311658,27.9483297927613],[0.00918827288987244,-0.000958205797942005,-0.994563756282914,-0.103718813005981],[0,0,0,0],[9E+09,9E+09,9E+09,9E+09,9E+09,9E+09]],
		[[292.368651285828,-233.880209617552,-21.7501213277837],[0.00918827288987244,-0.000958205797942005,-0.994563756282914,-0.103718813005981],[0,0,0,0],[9E+09,9E+09,9E+09,9E+09,9E+09,9E+09]],
		[[292.368651285828,-233.880209617552,-21.7501213277837],[0.00918827288987244,-0.000958205797942005,-0.994563756282914,-0.103718813005981],[0,0,0,0],[9E+09,9E+09,9E+09,9E+09,9E+09,9E+09]],
		[[291.794678644652,-227.329309808736,-52.8116532781243],[0.00918827288987244,-0.000958205797942005,-0.994563756282914,-0.103718813005981],[0,0,0,0],[9E+09,9E+09,9E+09,9E+09,9E+09,9E+09]],
		[[291.794678644652,-227.329309808736,-52.8116532781243],[0.00918827288987244,-0.000958205797942005,-0.994563756282914,-0.103718813005981],[0,0,0,0],[9E+09,9E+09,9E+09,9E+09,9E+09,9E+09]],
		[[292.368651285828,-233.880209617552,-21.7501213277837],[0.00918827288987244,-0.000958205797942005,-0.994563756282914,-0.103718813005981],[0,0,0,0],[9E+09,9E+09,9E+09,9E+09,9E+09,9E+09]],
		[[293.28700751171,-244.361649311658,27.9483297927613],[0.00918827288987244,-0.000958205797942005,-0.994563756282914,-0.103718813005981],[0,0,0,0],[9E+09,9E+09,9E+09,9E+09,9E+09,9E+09]],
		[[249.459094617476,-137.316682571751,46.0807019976294],[0.00720641123076419,-0.000415118187492874,-0.998318997016837,-0.0575071778942388],[0,0,0,0],[9E+09,9E+09,9E+09,9E+09,9E+09,9E+09]],
		[[248.730579441892,-131.483471005379,-4.37802280255641],[0.00720641123076419,-0.000415118187492874,-0.998318997016837,-0.0575071778942388],[0,0,0,0],[9E+09,9E+09,9E+09,9E+09,9E+09,9E+09]],
		[[248.730579441892,-131.483471005379,-4.37802280255641],[0.00720641123076419,-0.000415118187492874,-0.998318997016837,-0.0575071778942388],[0,0,0,0],[9E+09,9E+09,9E+09,9E+09,9E+09,9E+09]],
		[[248.275257457153,-127.837713776397,-35.9147258026727],[0.00720641123076419,-0.000415118187492874,-0.998318997016837,-0.0575071778942388],[0,0,0,0],[9E+09,9E+09,9E+09,9E+09,9E+09,9E+09]],
		[[248.275257457153,-127.837713776397,-35.9147258026727],[0.00720641123076419,-0.000415118187492874,-0.998318997016837,-0.0575071778942388],[0,0,0,0],[9E+09,9E+09,9E+09,9E+09,9E+09,9E+09]],
		[[248.730579441892,-131.483471005379,-4.37802280255641],[0.00720641123076419,-0.000415118187492874,-0.998318997016837,-0.0575071778942388],[0,0,0,0],[9E+09,9E+09,9E+09,9E+09,9E+09,9E+09]],
		[[249.459094617476,-137.316682571751,46.0807019976294],[0.00720641123076419,-0.000415118187492874,-0.998318997016837,-0.0575071778942388],[0,0,0,0],[9E+09,9E+09,9E+09,9E+09,9E+09,9E+09]],
		[[290.829543745998,-100.056182181525,49.234722450473],[0.00680707504627507,-0.000287946923608445,-0.999083317268074,-0.042262346982922],[0,0,0,0],[9E+09,9E+09,9E+09,9E+09,9E+09,9E+09]],
		[[290.139815300174,-95.7660646865366,-1.37910141761904],[0.00680707504627507,-0.000287946923608445,-0.999083317268074,-0.042262346982922],[0,0,0,0],[9E+09,9E+09,9E+09,9E+09,9E+09,9E+09]],
		[[290.139815300174,-95.7660646865366,-1.37910141761904],[0.00680707504627507,-0.000287946923608445,-0.999083317268074,-0.042262346982922],[0,0,0,0],[9E+09,9E+09,9E+09,9E+09,9E+09,9E+09]],
		[[289.708735021536,-93.0847412521693,-33.0127413351765],[0.00680707504627507,-0.000287946923608445,-0.999083317268074,-0.042262346982922],[0,0,0,0],[9E+09,9E+09,9E+09,9E+09,9E+09,9E+09]],
		[[289.708735021536,-93.0847412521693,-33.0127413351765],[0.00680707504627507,-0.000287946923608445,-0.999083317268074,-0.042262346982922],[0,0,0,0],[9E+09,9E+09,9E+09,9E+09,9E+09,9E+09]],
		[[290.139815300174,-95.7660646865366,-1.37910141761904],[0.00680707504627507,-0.000287946923608445,-0.999083317268074,-0.042262346982922],[0,0,0,0],[9E+09,9E+09,9E+09,9E+09,9E+09,9E+09]],
		[[290.829543745998,-100.056182181525,49.234722450473],[0.00680707504627507,-0.000287946923608445,-0.999083317268074,-0.042262346982922],[0,0,0,0],[9E+09,9E+09,9E+09,9E+09,9E+09,9E+09]],
		[[245.740187119161,-87.6128069534354,50.8276032034953],[0.0066909782554097,-0.000245268224154555,-0.999306424862602,-0.0366311326852939],[0,0,0,0],[9E+09,9E+09,9E+09,9E+09,9E+09,9E+09]],
		[[245.061768043552,-83.8934984330366,0.16848268519243],[0.0066909782554097,-0.000245268224154555,-0.999306424862602,-0.0366311326852939],[0,0,0,0],[9E+09,9E+09,9E+09,9E+09,9E+09,9E+09]],
		[[245.061768043552,-83.8934984330366,0.16848268519243],[0.0066909782554097,-0.000245268224154555,-0.999306424862602,-0.0366311326852939],[0,0,0,0],[9E+09,9E+09,9E+09,9E+09,9E+09,9E+09]],
		[[244.637756121297,-81.5689306077871,-31.493467638747],[0.0066909782554097,-0.000245268224154555,-0.999306424862602,-0.0366311326852939],[0,0,0,0],[9E+09,9E+09,9E+09,9E+09,9E+09,9E+09]],
		[[244.637756121297,-81.5689306077871,-31.493467638747],[0.0066909782554097,-0.000245268224154555,-0.999306424862602,-0.0366311326852939],[0,0,0,0],[9E+09,9E+09,9E+09,9E+09,9E+09,9E+09]],
		[[245.061768043552,-83.8934984330366,0.16848268519243],[0.0066909782554097,-0.000245268224154555,-0.999306424862602,-0.0366311326852939],[0,0,0,0],[9E+09,9E+09,9E+09,9E+09,9E+09,9E+09]],
		[[245.740187119161,-87.6128069534354,50.8276032034953],[0.0066909782554097,-0.000245268224154555,-0.999306424862602,-0.0366311326852939],[0,0,0,0],[9E+09,9E+09,9E+09,9E+09,9E+09,9E+09]],
		[[403.099233829671,-245.749127372575,25.6017542319324],[0.00936954043940217,-0.00100794170503457,-0.994219250722917,-0.106954556973674],[0,0,0,0],[9E+09,9E+09,9E+09,9E+09,9E+09,9E+09]],
		[[402.163744360367,-234.944401870427,-24.0270959086467],[0.00936954043940217,-0.00100794170503457,-0.994219250722917,-0.106954556973674],[0,0,0,0],[9E+09,9E+09,9E+09,9E+09,9E+09,9E+09]],
		[[402.163744360367,-234.944401870427,-24.0270959086467],[0.00936954043940217,-0.00100794170503457,-0.994219250722917,-0.106954556973674],[0,0,0,0],[9E+09,9E+09,9E+09,9E+09,9E+09,9E+09]],
		[[401.579063442052,-228.191448431585,-55.0451272465088],[0.00936954043940217,-0.00100794170503457,-0.994219250722917,-0.106954556973674],[0,0,0,0],[9E+09,9E+09,9E+09,9E+09,9E+09,9E+09]],
		[[401.579063442052,-228.191448431585,-55.0451272465088],[0.00936954043940217,-0.00100794170503457,-0.994219250722917,-0.106954556973674],[0,0,0,0],[9E+09,9E+09,9E+09,9E+09,9E+09,9E+09]],
		[[402.163744360367,-234.944401870427,-24.0270959086467],[0.00936954043940217,-0.00100794170503457,-0.994219250722917,-0.106954556973674],[0,0,0,0],[9E+09,9E+09,9E+09,9E+09,9E+09,9E+09]],
		[[403.099233829671,-245.749127372575,25.6017542319324],[0.00936954043940217,-0.00100794170503457,-0.994219250722917,-0.106954556973674],[0,0,0,0],[9E+09,9E+09,9E+09,9E+09,9E+09,9E+09]],
		[[396.033748937128,-194.18703812988,35.7216135201404],[0.00820516010917249,-0.000693329099167655,-0.996415168384063,-0.0841962401565701],[0,0,0,0],[9E+09,9E+09,9E+09,9E+09,9E+09,9E+09]],
		[[395.209024115822,-185.662788001459,-14.3513031985533],[0.00820516010917249,-0.000693329099167655,-0.996415168384063,-0.0841962401565701],[0,0,0,0],[9E+09,9E+09,9E+09,9E+09,9E+09,9E+09]],
		[[395.209024115822,-185.662788001459,-14.3513031985533],[0.00820516010917249,-0.000693329099167655,-0.996415168384063,-0.0841962401565701],[0,0,0,0],[9E+09,9E+09,9E+09,9E+09,9E+09,9E+09]],
		[[394.693571102503,-180.335131671196,-45.6468761477369],[0.00820516010917249,-0.000693329099167655,-0.996415168384063,-0.0841962401565701],[0,0,0,0],[9E+09,9E+09,9E+09,9E+09,9E+09,9E+09]],
		[[394.693571102503,-180.335131671196,-45.6468761477369],[0.00820516010917249,-0.000693329099167655,-0.996415168384063,-0.0841962401565701],[0,0,0,0],[9E+09,9E+09,9E+09,9E+09,9E+09,9E+09]],
		[[395.209024115822,-185.662788001459,-14.3513031985533],[0.00820516010917249,-0.000693329099167655,-0.996415168384063,-0.0841962401565701],[0,0,0,0],[9E+09,9E+09,9E+09,9E+09,9E+09,9E+09]],
		[[396.033748937128,-194.18703812988,35.7216135201404],[0.00820516010917249,-0.000693329099167655,-0.996415168384063,-0.0841962401565701],[0,0,0,0],[9E+09,9E+09,9E+09,9E+09,9E+09,9E+09]],
		[[391.06989532529,-137.544241837855,44.000996564666],[0.00726571628808549,-0.000432828028158066,-0.998203897421597,-0.0594642850714026],[0,0,0,0],[9E+09,9E+09,9E+09,9E+09,9E+09,9E+09]],
		[[390.335639388971,-131.51320224425,-6.43438218517918],[0.00726571628808549,-0.000432828028158066,-0.998203897421597,-0.0594642850714026],[0,0,0,0],[9E+09,9E+09,9E+09,9E+09,9E+09,9E+09]],
		[[390.335639388971,-131.51320224425,-6.43438218517918],[0.00726571628808549,-0.000432828028158066,-0.998203897421597,-0.0594642850714026],[0,0,0,0],[9E+09,9E+09,9E+09,9E+09,9E+09,9E+09]],
		[[389.876729428771,-127.743802498246,-37.9564939038324],[0.00726571628808549,-0.000432828028158066,-0.998203897421597,-0.0594642850714026],[0,0,0,0],[9E+09,9E+09,9E+09,9E+09,9E+09,9E+09]],
		[[389.876729428771,-127.743802498246,-37.9564939038324],[0.00726571628808549,-0.000432828028158066,-0.998203897421597,-0.0594642850714026],[0,0,0,0],[9E+09,9E+09,9E+09,9E+09,9E+09,9E+09]],
		[[390.335639388971,-131.51320224425,-6.43438218517918],[0.00726571628808549,-0.000432828028158066,-0.998203897421597,-0.0594642850714026],[0,0,0,0],[9E+09,9E+09,9E+09,9E+09,9E+09,9E+09]],
		[[391.06989532529,-137.544241837855,44.000996564666],[0.00726571628808549,-0.000432828028158066,-0.998203897421597,-0.0594642850714026],[0,0,0,0],[9E+09,9E+09,9E+09,9E+09,9E+09,9E+09]],
		[[385.668546901666,-85.4729115296458,49.1107245728777],[0.00669526575096486,-0.000247046366600005,-0.999297509827073,-0.0368727438364299],[0,0,0,0],[9E+09,9E+09,9E+09,9E+09,9E+09,9E+09]],
		[[384.989711265164,-81.7291044236946,-1.54658576365773],[0.00669526575096486,-0.000247046366600005,-0.999297509827073,-0.0368727438364299],[0,0,0,0],[9E+09,9E+09,9E+09,9E+09,9E+09,9E+09]],
		[[384.989711265164,-81.7291044236946,-1.54658576365773],[0.00669526575096486,-0.000247046366600005,-0.999297509827073,-0.0368727438364299],[0,0,0,0],[9E+09,9E+09,9E+09,9E+09,9E+09,9E+09]],
		[[384.565438992351,-79.389224982475,-33.2074047239924],[0.00669526575096486,-0.000247046366600005,-0.999297509827073,-0.0368727438364299],[0,0,0,0],[9E+09,9E+09,9E+09,9E+09,9E+09,9E+09]],
		[[384.565438992351,-79.389224982475,-33.2074047239924],[0.00669526575096486,-0.000247046366600005,-0.999297509827073,-0.0368727438364299],[0,0,0,0],[9E+09,9E+09,9E+09,9E+09,9E+09,9E+09]],
		[[384.989711265164,-81.7291044236946,-1.54658576365773],[0.00669526575096486,-0.000247046366600005,-0.999297509827073,-0.0368727438364299],[0,0,0,0],[9E+09,9E+09,9E+09,9E+09,9E+09,9E+09]],
		[[385.668546901666,-85.4729115296458,49.1107245728777],[0.00669526575096486,-0.000247046366600005,-0.999297509827073,-0.0368727438364299],[0,0,0,0],[9E+09,9E+09,9E+09,9E+09,9E+09,9E+09]],
		[[478.315791276222,-86.4437658870823,47.794069485851],[0.00671892774812616,-0.000256146261682229,-0.999251517650421,-0.038094551740885],[0,0,0,0],[9E+09,9E+09,9E+09,9E+09,9E+09,9E+09]],
		[[477.634650553439,-82.5760815046593,-2.85390248572684],[0.00671892774812616,-0.000256146261682229,-0.999251517650421,-0.038094551740885],[0,0,0,0],[9E+09,9E+09,9E+09,9E+09,9E+09,9E+09]],
		[[477.634650553439,-82.5760815046593,-2.85390248572684],[0.00671892774812616,-0.000256146261682229,-0.999251517650421,-0.038094551740885],[0,0,0,0],[9E+09,9E+09,9E+09,9E+09,9E+09,9E+09]],
		[[477.208937601699,-80.1587787656448,-34.5088849679627],[0.00671892774812616,-0.000256146261682229,-0.999251517650421,-0.038094551740885],[0,0,0,0],[9E+09,9E+09,9E+09,9E+09,9E+09,9E+09]],
		[[477.208937601699,-80.1587787656448,-34.5088849679627],[0.00671892774812616,-0.000256146261682229,-0.999251517650421,-0.038094551740885],[0,0,0,0],[9E+09,9E+09,9E+09,9E+09,9E+09,9E+09]],
		[[477.634650553439,-82.5760815046593,-2.85390248572684],[0.00671892774812616,-0.000256146261682229,-0.999251517650421,-0.038094551740885],[0,0,0,0],[9E+09,9E+09,9E+09,9E+09,9E+09,9E+09]],
		[[478.315791276222,-86.4437658870823,47.794069485851],[0.00671892774812616,-0.000256146261682229,-0.999251517650421,-0.038094551740885],[0,0,0,0],[9E+09,9E+09,9E+09,9E+09,9E+09,9E+09]],
		[[483.133106013849,-138.756801668918,42.5082331765351],[0.0073226084519266,-0.000449565472182051,-0.998093827794076,-0.0612771426856401],[0,0,0,0],[9E+09,9E+09,9E+09,9E+09,9E+09,9E+09]],
		[[482.393346029146,-132.54257687196,-7.904822328343],[0.0073226084519266,-0.000449565472182051,-0.998093827794076,-0.0612771426856401],[0,0,0,0],[9E+09,9E+09,9E+09,9E+09,9E+09,9E+09]],
		[[482.393346029146,-132.54257687196,-7.904822328343],[0.0073226084519266,-0.000449565472182051,-0.998093827794076,-0.0612771426856401],[0,0,0,0],[9E+09,9E+09,9E+09,9E+09,9E+09,9E+09]],
		[[481.930996038706,-128.658686373861,-39.4129820188915],[0.0073226084519266,-0.000449565472182051,-0.998093827794076,-0.0612771426856401],[0,0,0,0],[9E+09,9E+09,9E+09,9E+09,9E+09,9E+09]],
		[[481.930996038706,-128.658686373861,-39.4129820188915],[0.0073226084519266,-0.000449565472182051,-0.998093827794076,-0.0612771426856401],[0,0,0,0],[9E+09,9E+09,9E+09,9E+09,9E+09,9E+09]],
		[[482.393346029146,-132.54257687196,-7.904822328343],[0.0073226084519266,-0.000449565472182051,-0.998093827794076,-0.0612771426856401],[0,0,0,0],[9E+09,9E+09,9E+09,9E+09,9E+09,9E+09]],
		[[483.133106013849,-138.756801668918,42.5082331765351],[0.0073226084519266,-0.000449565472182051,-0.998093827794076,-0.0612771426856401],[0,0,0,0],[9E+09,9E+09,9E+09,9E+09,9E+09,9E+09]],
		[[483.222642292122,-189.861338067738,35.0219683114554],[0.00819448846874309,-0.000690679339774657,-0.996433068445667,-0.0839851976763621],[0,0,0,0],[9E+09,9E+09,9E+09,9E+09,9E+09,9E+09]],
		[[482.39894544337,-181.3583032081,-15.0545723206324],[0.00819448846874309,-0.000690679339774657,-0.996433068445667,-0.0839851976763621],[0,0,0,0],[9E+09,9E+09,9E+09,9E+09,9E+09,9E+09]],
		[[482.39894544337,-181.3583032081,-15.0545723206324],[0.00819448846874309,-0.000690679339774657,-0.996433068445667,-0.0839851976763621],[0,0,0,0],[9E+09,9E+09,9E+09,9E+09,9E+09,9E+09]],
		[[481.884134912899,-176.043906420827,-46.3524102156873],[0.00819448846874309,-0.000690679339774657,-0.996433068445667,-0.0839851976763621],[0,0,0,0],[9E+09,9E+09,9E+09,9E+09,9E+09,9E+09]],
		[[481.884134912899,-176.043906420827,-46.3524102156873],[0.00819448846874309,-0.000690679339774657,-0.996433068445667,-0.0839851976763621],[0,0,0,0],[9E+09,9E+09,9E+09,9E+09,9E+09,9E+09]],
		[[482.39894544337,-181.3583032081,-15.0545723206324],[0.00819448846874309,-0.000690679339774657,-0.996433068445667,-0.0839851976763621],[0,0,0,0],[9E+09,9E+09,9E+09,9E+09,9E+09,9E+09]],
		[[483.222642292122,-189.861338067738,35.0219683114554],[0.00819448846874309,-0.000690679339774657,-0.996433068445667,-0.0839851976763621],[0,0,0,0],[9E+09,9E+09,9E+09,9E+09,9E+09,9E+09]],
		[[489.630453604917,-244.907439108101,24.1464954374401],[0.00947203461223947,-0.00103629582389185,-0.994023250292104,-0.108751940350465],[0,0,0,0],[9E+09,9E+09,9E+09,9E+09,9E+09,9E+09]],
		[[488.685296902346,-233.923282965952,-25.4427674392399],[0.00947203461223947,-0.00103629582389185,-0.994023250292104,-0.108751940350465],[0,0,0,0],[9E+09,9E+09,9E+09,9E+09,9E+09,9E+09]],
		[[488.685296902346,-233.923282965952,-25.4427674392399],[0.00947203461223947,-0.00103629582389185,-0.994023250292104,-0.108751940350465],[0,0,0,0],[9E+09,9E+09,9E+09,9E+09,9E+09,9E+09]],
		[[488.094573963238,-227.058185377108,-56.4360567371645],[0.00947203461223947,-0.00103629582389185,-0.994023250292104,-0.108751940350465],[0,0,0,0],[9E+09,9E+09,9E+09,9E+09,9E+09,9E+09]],
		[[488.094573963238,-227.058185377108,-56.4360567371645],[0.00947203461223947,-0.00103629582389185,-0.994023250292104,-0.108751940350465],[0,0,0,0],[9E+09,9E+09,9E+09,9E+09,9E+09,9E+09]],
		[[488.685296902346,-233.923282965952,-25.4427674392399],[0.00947203461223947,-0.00103629582389185,-0.994023250292104,-0.108751940350465],[0,0,0,0],[9E+09,9E+09,9E+09,9E+09,9E+09,9E+09]],
		[[489.630453604917,-244.907439108101,24.1464954374401],[0.00947203461223947,-0.00103629582389185,-0.994023250292104,-0.108751940350465],[0,0,0,0],[9E+09,9E+09,9E+09,9E+09,9E+09,9E+09]],
		[[602.136376955429,-240.655233611394,22.9421139308661],[0.00952750400653266,-0.0010519700999858,-0.993913882382944,-0.109742035851254],[0,0,0,0],[9E+09,9E+09,9E+09,9E+09,9E+09,9E+09]],
		[[601.186003122767,-229.572283406206,-26.6250627521719],[0.00952750400653266,-0.0010519700999858,-0.993913882382944,-0.109742035851254],[0,0,0,0],[9E+09,9E+09,9E+09,9E+09,9E+09,9E+09]],
		[[601.186003122767,-229.572283406206,-26.6250627521719],[0.00952750400653266,-0.0010519700999858,-0.993913882382944,-0.109742035851254],[0,0,0,0],[9E+09,9E+09,9E+09,9E+09,9E+09,9E+09]],
		[[600.592019477353,-222.645439527964,-57.604548179071],[0.00952750400653266,-0.0010519700999858,-0.993913882382944,-0.109742035851254],[0,0,0,0],[9E+09,9E+09,9E+09,9E+09,9E+09,9E+09]],
		[[600.592019477353,-222.645439527964,-57.604548179071],[0.00952750400653266,-0.0010519700999858,-0.993913882382944,-0.109742035851254],[0,0,0,0],[9E+09,9E+09,9E+09,9E+09,9E+09,9E+09]],
		[[601.186003122767,-229.572283406206,-26.6250627521719],[0.00952750400653266,-0.0010519700999858,-0.993913882382944,-0.109742035851254],[0,0,0,0],[9E+09,9E+09,9E+09,9E+09,9E+09,9E+09]],
		[[602.136376955429,-240.655233611394,22.9421139308661],[0.00952750400653266,-0.0010519700999858,-0.993913882382944,-0.109742035851254],[0,0,0,0],[9E+09,9E+09,9E+09,9E+09,9E+09,9E+09]],
		[[594.105058195658,-186.41205556819,33.7829943400776],[0.00822215146796232,-0.000698454025213563,-0.996377418391712,-0.0846401116863593],[0,0,0,0],[9E+09,9E+09,9E+09,9E+09,9E+09,9E+09]],
		[[593.278720114878,-177.843188909236,-16.2822799481687],[0.00822215146796232,-0.000698454025213563,-0.996377418391712,-0.0846401116863593],[0,0,0,0],[9E+09,9E+09,9E+09,9E+09,9E+09,9E+09]],
		[[593.278720114878,-177.843188909236,-16.2822799481687],[0.00822215146796232,-0.000698454025213563,-0.996377418391712,-0.0846401116863593],[0,0,0,0],[9E+09,9E+09,9E+09,9E+09,9E+09,9E+09]],
		[[592.762258814391,-172.48764724739,-47.5730763783227],[0.00822215146796232,-0.000698454025213563,-0.996377418391712,-0.0846401116863593],[0,0,0,0],[9E+09,9E+09,9E+09,9E+09,9E+09,9E+09]],
		[[592.762258814391,-172.48764724739,-47.5730763783227],[0.00822215146796232,-0.000698454025213563,-0.996377418391712,-0.0846401116863593],[0,0,0,0],[9E+09,9E+09,9E+09,9E+09,9E+09,9E+09]],
		[[593.278720114878,-177.843188909236,-16.2822799481687],[0.00822215146796232,-0.000698454025213563,-0.996377418391712,-0.0846401116863593],[0,0,0,0],[9E+09,9E+09,9E+09,9E+09,9E+09,9E+09]],
		[[594.105058195658,-186.41205556819,33.7829943400776],[0.00822215146796232,-0.000698454025213563,-0.996377418391712,-0.0846401116863593],[0,0,0,0],[9E+09,9E+09,9E+09,9E+09,9E+09,9E+09]],
		[[594.013579836482,-136.119059315104,41.2060164577616],[0.00733540540573417,-0.000453473807444863,-0.99806765566097,-0.0617004125792975],[0,0,0,0],[9E+09,9E+09,9E+09,9E+09,9E+09,9E+09]],
		[[593.272585498753,-129.862072839968,-9.20173143521038],[0.00733540540573417,-0.000453473807444863,-0.99806765566097,-0.0617004125792975],[0,0,0,0],[9E+09,9E+09,9E+09,9E+09,9E+09,9E+09]],
		[[593.272585498753,-129.862072839968,-9.20173143521038],[0.00733540540573417,-0.000453473807444863,-0.99806765566097,-0.0617004125792975],[0,0,0,0],[9E+09,9E+09,9E+09,9E+09,9E+09,9E+09]],
		[[592.809464037672,-125.951456293008,-40.7065738683178],[0.00733540540573417,-0.000453473807444863,-0.99806765566097,-0.0617004125792975],[0,0,0,0],[9E+09,9E+09,9E+09,9E+09,9E+09,9E+09]],
		[[592.809464037672,-125.951456293008,-40.7065738683178],[0.00733540540573417,-0.000453473807444863,-0.99806765566097,-0.0617004125792975],[0,0,0,0],[9E+09,9E+09,9E+09,9E+09,9E+09,9E+09]],
		[[593.272585498753,-129.862072839968,-9.20173143521038],[0.00733540540573417,-0.000453473807444863,-0.99806765566097,-0.0617004125792975],[0,0,0,0],[9E+09,9E+09,9E+09,9E+09,9E+09,9E+09]],
		[[594.013579836482,-136.119059315104,41.2060164577616],[0.00733540540573417,-0.000453473807444863,-0.99806765566097,-0.0617004125792975],[0,0,0,0],[9E+09,9E+09,9E+09,9E+09,9E+09,9E+09]],
		[[593.951420595743,-86.0463664067457,46.2676477594915],[0.00673606385428096,-0.000262673005791383,-0.999217855075423,-0.0389645293198063],[0,0,0,0],[9E+09,9E+09,9E+09,9E+09,9E+09,9E+09]],
		[[593.268611664579,-82.090486810967,-4.37348955581023],[0.00673606385428096,-0.000262673005791383,-0.999217855075423,-0.0389645293198063],[0,0,0,0],[9E+09,9E+09,9E+09,9E+09,9E+09,9E+09]],
		[[593.268611664579,-82.090486810967,-4.37348955581023],[0.00673606385428096,-0.000262673005791383,-0.999217855075423,-0.0389645293198063],[0,0,0,0],[9E+09,9E+09,9E+09,9E+09,9E+09,9E+09]],
		[[592.841856082603,-79.6180620636052,-36.0242003778737],[0.00673606385428096,-0.000262673005791383,-0.999217855075423,-0.0389645293198063],[0,0,0,0],[9E+09,9E+09,9E+09,9E+09,9E+09,9E+09]],
		[[592.841856082603,-79.6180620636052,-36.0242003778737],[0.00673606385428096,-0.000262673005791383,-0.999217855075423,-0.0389645293198063],[0,0,0,0],[9E+09,9E+09,9E+09,9E+09,9E+09,9E+09]],
		[[593.268611664579,-82.090486810967,-4.37348955581023],[0.00673606385428096,-0.000262673005791383,-0.999217855075423,-0.0389645293198063],[0,0,0,0],[9E+09,9E+09,9E+09,9E+09,9E+09,9E+09]],
		[[593.951420595743,-86.0463664067457,46.2676477594915],[0.00673606385428096,-0.000262673005791383,-0.999217855075423,-0.0389645293198063],[0,0,0,0],[9E+09,9E+09,9E+09,9E+09,9E+09,9E+09]]
		];

	!Speeds
	CONST speeddata WorkingstepSpeeddatas{140} := [
		[ 800, 500, 5000, 1000],
		[ 800, 500, 5000, 1000],
		[ 4.23333333333333, 500, 5000, 1000],
		[ 4.23333333333333, 500, 5000, 1000],
		[ 800, 500, 5000, 1000],
		[ 800, 500, 5000, 1000],
		[ 800, 500, 5000, 1000],
		[ 800, 500, 5000, 1000],
		[ 800, 500, 5000, 1000],
		[ 4.23333333333333, 500, 5000, 1000],
		[ 4.23333333333333, 500, 5000, 1000],
		[ 800, 500, 5000, 1000],
		[ 800, 500, 5000, 1000],
		[ 800, 500, 5000, 1000],
		[ 800, 500, 5000, 1000],
		[ 800, 500, 5000, 1000],
		[ 4.23333333333333, 500, 5000, 1000],
		[ 4.23333333333333, 500, 5000, 1000],
		[ 800, 500, 5000, 1000],
		[ 800, 500, 5000, 1000],
		[ 800, 500, 5000, 1000],
		[ 800, 500, 5000, 1000],
		[ 800, 500, 5000, 1000],
		[ 4.23333333333333, 500, 5000, 1000],
		[ 4.23333333333333, 500, 5000, 1000],
		[ 800, 500, 5000, 1000],
		[ 800, 500, 5000, 1000],
		[ 800, 500, 5000, 1000],
		[ 800, 500, 5000, 1000],
		[ 800, 500, 5000, 1000],
		[ 4.23333333333333, 500, 5000, 1000],
		[ 4.23333333333333, 500, 5000, 1000],
		[ 800, 500, 5000, 1000],
		[ 800, 500, 5000, 1000],
		[ 800, 500, 5000, 1000],
		[ 800, 500, 5000, 1000],
		[ 800, 500, 5000, 1000],
		[ 4.23333333333333, 500, 5000, 1000],
		[ 4.23333333333333, 500, 5000, 1000],
		[ 800, 500, 5000, 1000],
		[ 800, 500, 5000, 1000],
		[ 800, 500, 5000, 1000],
		[ 800, 500, 5000, 1000],
		[ 800, 500, 5000, 1000],
		[ 4.23333333333333, 500, 5000, 1000],
		[ 4.23333333333333, 500, 5000, 1000],
		[ 800, 500, 5000, 1000],
		[ 800, 500, 5000, 1000],
		[ 800, 500, 5000, 1000],
		[ 800, 500, 5000, 1000],
		[ 800, 500, 5000, 1000],
		[ 4.23333333333333, 500, 5000, 1000],
		[ 4.23333333333333, 500, 5000, 1000],
		[ 800, 500, 5000, 1000],
		[ 800, 500, 5000, 1000],
		[ 800, 500, 5000, 1000],
		[ 800, 500, 5000, 1000],
		[ 800, 500, 5000, 1000],
		[ 4.23333333333333, 500, 5000, 1000],
		[ 4.23333333333333, 500, 5000, 1000],
		[ 800, 500, 5000, 1000],
		[ 800, 500, 5000, 1000],
		[ 800, 500, 5000, 1000],
		[ 800, 500, 5000, 1000],
		[ 800, 500, 5000, 1000],
		[ 4.23333333333333, 500, 5000, 1000],
		[ 4.23333333333333, 500, 5000, 1000],
		[ 800, 500, 5000, 1000],
		[ 800, 500, 5000, 1000],
		[ 800, 500, 5000, 1000],
		[ 800, 500, 5000, 1000],
		[ 800, 500, 5000, 1000],
		[ 4.23333333333333, 500, 5000, 1000],
		[ 4.23333333333333, 500, 5000, 1000],
		[ 800, 500, 5000, 1000],
		[ 800, 500, 5000, 1000],
		[ 800, 500, 5000, 1000],
		[ 800, 500, 5000, 1000],
		[ 800, 500, 5000, 1000],
		[ 4.23333333333333, 500, 5000, 1000],
		[ 4.23333333333333, 500, 5000, 1000],
		[ 800, 500, 5000, 1000],
		[ 800, 500, 5000, 1000],
		[ 800, 500, 5000, 1000],
		[ 800, 500, 5000, 1000],
		[ 800, 500, 5000, 1000],
		[ 4.23333333333333, 500, 5000, 1000],
		[ 4.23333333333333, 500, 5000, 1000],
		[ 800, 500, 5000, 1000],
		[ 800, 500, 5000, 1000],
		[ 800, 500, 5000, 1000],
		[ 800, 500, 5000, 1000],
		[ 800, 500, 5000, 1000],
		[ 4.23333333333333, 500, 5000, 1000],
		[ 4.23333333333333, 500, 5000, 1000],
		[ 800, 500, 5000, 1000],
		[ 800, 500, 5000, 1000],
		[ 800, 500, 5000, 1000],
		[ 800, 500, 5000, 1000],
		[ 800, 500, 5000, 1000],
		[ 4.23333333333333, 500, 5000, 1000],
		[ 4.23333333333333, 500, 5000, 1000],
		[ 800, 500, 5000, 1000],
		[ 800, 500, 5000, 1000],
		[ 800, 500, 5000, 1000],
		[ 800, 500, 5000, 1000],
		[ 800, 500, 5000, 1000],
		[ 4.23333333333333, 500, 5000, 1000],
		[ 4.23333333333333, 500, 5000, 1000],
		[ 800, 500, 5000, 1000],
		[ 800, 500, 5000, 1000],
		[ 800, 500, 5000, 1000],
		[ 800, 500, 5000, 1000],
		[ 800, 500, 5000, 1000],
		[ 4.23333333333333, 500, 5000, 1000],
		[ 4.23333333333333, 500, 5000, 1000],
		[ 800, 500, 5000, 1000],
		[ 800, 500, 5000, 1000],
		[ 800, 500, 5000, 1000],
		[ 800, 500, 5000, 1000],
		[ 800, 500, 5000, 1000],
		[ 4.23333333333333, 500, 5000, 1000],
		[ 4.23333333333333, 500, 5000, 1000],
		[ 800, 500, 5000, 1000],
		[ 800, 500, 5000, 1000],
		[ 800, 500, 5000, 1000],
		[ 800, 500, 5000, 1000],
		[ 800, 500, 5000, 1000],
		[ 4.23333333333333, 500, 5000, 1000],
		[ 4.23333333333333, 500, 5000, 1000],
		[ 800, 500, 5000, 1000],
		[ 800, 500, 5000, 1000],
		[ 800, 500, 5000, 1000],
		[ 800, 500, 5000, 1000],
		[ 800, 500, 5000, 1000],
		[ 4.23333333333333, 500, 5000, 1000],
		[ 4.23333333333333, 500, 5000, 1000],
		[ 800, 500, 5000, 1000],
		[ 800, 500, 5000, 1000],
		[ 800, 500, 5000, 1000]
		];


ENDMODULE

--- Backups/Rob1/RAPID/TASK1/PROGMOD/StanWorkingPlan.mod ---
MODULE StanWorkingPlan

    RECORD msgrec
        string controllerName;
        string workStep;
        string featureName;
        string featureUUID;
    ENDRECORD

    PERS string msgSlot:="Stan";
    PERS string previousUUID:="c5793a88-d117-412a-8380-89480e2aa149";



    PERS string workingPlanUUID:="sdvonvskvnwovewn342532nkfloencvosnvqwef12";
    PERS string AP238_WORKINGSTEP_NAME := "";
    PERS string AP238_WORKINGSTEP_UUID := "";
    PERS string AP238_FEATURE_NAME := "";
    PERS string AP238_FEATURE_UUID := "";
    PERS bool ok;
    PERS num startIndex :=134;
    PERS num stopIndex :=140;
      CONST speeddata serge := [ 800, 500, 5000, 1000];



    PROC main()
        AP238_WORKINGSTEP_NAME := "";

       !  SetDO IsDone,0;
         MoveAbsJ jHome,v400,z10,PendEff_point\WObj:=A;
        MoveAbsJ jee,v400,z10,PendEff_point\WObj:=A;
        ConfJ\Off;
        ConfL\Off;

       FOR i FROM 1 TO dim(WorkPlan,1) DO

           ok := StrToVal(Workplan{i,1}, startIndex);
           ok := StrToVal(Workplan{i,2}, stopIndex);

                WorkingStep startIndex, stopIndex, Workplan{i,3}, Workplan{i,4}, Workplan{i,5}, Workplan{i,6}, WorkingstepRobtargets, WorkingstepSpeeddatas;

        ENDFOR

        MoveAbsJ jee,v400,z10,PendEff_point\WObj:=A;
        MoveAbsJ jHome,v400,z10,PendEff_point\WObj:=A;
        AP238_WORKINGSTEP_NAME := "";
    ENDPROC

    PROC WorkingStep(num startpos, num endpos, string workingstepName, string workingstepUUID, string featureName, string featureUUID, robtarget targetList{*}, speeddata speedList{*})
      VAR msgrec data;

        FOR i FROM startpos TO endpos DO

      !           SetDO IsDone,0;



            AP238_WORKINGSTEP_NAME := workingstepName;

            !send message
            data.controllerName := msgSlot;
            data.workStep := workingstepName;
            data.featureName := featureName;
            data.featureUUID := featureUUID;
            !sendMessage data, msgSlot;

            AP238_WORKINGSTEP_UUID := workingstepUUID;
            AP238_FEATURE_NAME := featureName;
            AP238_FEATURE_UUID := featureUUID;
     !       MoveL targetList{i},v1000,z100,PendEff_point\WObj:=A;
            MoveL Workingsteprobtargets{i}, speedList{i}, z100,PendEff_point\WObj:=A;
     !       SetDO IsDone,1;
            AP238_WORKINGSTEP_NAME := "";
            AP238_WORKINGSTEP_UUID := "";
            AP238_FEATURE_NAME := "";
            AP238_FEATURE_UUID := "";
        ENDFOR

    ENDPROC

    PROC sendMessage(msgrec msg, string slot)
        VAR rmqslot myslot;
        IF previousUUID <> msg.featureUUID THEN
            RMQFindSlot myslot, slot;
            RMQSendMessage myslot, msg;
            previousUUID := msg.featureUUID;
        ENDIF
    ENDPROC


ENDMODULE

--- Backups/Rob1/RAPID/TASK1/SYSMOD/Speeds.sys ---
MODULE Speeds(SYSMODULE)
    !Rapid velocity
    VAR speeddata vRapid:=[800,500,5000,1000];

    VAR speeddata v0:=[800,500,5000,1000];
    VAR speeddata v1:=[800,500,5000,1000];
    VAR speeddata v2:=[4,500,5000,1000];
    VAR speeddata v3:=[4,500,5000,1000];
    VAR speeddata v4:=[800,500,5000,1000];
    VAR speeddata v5:=[800,500,5000,1000];
    VAR speeddata v6:=[800,500,5000,1000];
    VAR speeddata v7:=[800,500,5000,1000];
    VAR speeddata v8:=[800,500,5000,1000];
    VAR speeddata v9:=[4,500,5000,1000];
    VAR speeddata v10:=[4,500,5000,1000];
    VAR speeddata v11:=[800,500,5000,1000];
    VAR speeddata v12:=[800,500,5000,1000];
    VAR speeddata v13:=[800,500,5000,1000];
    VAR speeddata v14:=[800,500,5000,1000];
    VAR speeddata v15:=[800,500,5000,1000];
    VAR speeddata v16:=[4,500,5000,1000];
    VAR speeddata v17:=[4,500,5000,1000];
    VAR speeddata v18:=[800,500,5000,1000];
    VAR speeddata v19:=[800,500,5000,1000];
    VAR speeddata v20:=[800,500,5000,1000];
    VAR speeddata v21:=[800,500,5000,1000];
    VAR speeddata v22:=[800,500,5000,1000];
    VAR speeddata v23:=[4,500,5000,1000];
    VAR speeddata v24:=[4,500,5000,1000];
    VAR speeddata v25:=[800,500,5000,1000];
    VAR speeddata v26:=[800,500,5000,1000];
    VAR speeddata v27:=[800,500,5000,1000];
    VAR speeddata v28:=[800,500,5000,1000];
    VAR speeddata v29:=[800,500,5000,1000];
    VAR speeddata v30:=[4,500,5000,1000];
    VAR speeddata v31:=[4,500,5000,1000];
    VAR speeddata v32:=[800,500,5000,1000];
    VAR speeddata v33:=[800,500,5000,1000];
    VAR speeddata v34:=[800,500,5000,1000];
    VAR speeddata v35:=[800,500,5000,1000];
    VAR speeddata v36:=[800,500,5000,1000];
    VAR speeddata v37:=[4,500,5000,1000];
    VAR speeddata v38:=[4,500,5000,1000];
    VAR speeddata v39:=[800,500,5000,1000];
    VAR speeddata v40:=[800,500,5000,1000];
    VAR speeddata v41:=[800,500,5000,1000];
    VAR speeddata v42:=[800,500,5000,1000];
    VAR speeddata v43:=[800,500,5000,1000];
    VAR speeddata v44:=[4,500,5000,1000];
    VAR speeddata v45:=[4,500,5000,1000];
    VAR speeddata v46:=[800,500,5000,1000];
    VAR speeddata v47:=[800,500,5000,1000];
    VAR speeddata v48:=[800,500,5000,1000];
    VAR speeddata v49:=[800,500,5000,1000];
    VAR speeddata v50:=[800,500,5000,1000];
    VAR speeddata v51:=[4,500,5000,1000];
    VAR speeddata v52:=[4,500,5000,1000];
    VAR speeddata v53:=[800,500,5000,1000];
    VAR speeddata v54:=[800,500,5000,1000];
    VAR speeddata v55:=[800,500,5000,1000];
    VAR speeddata v56:=[800,500,5000,1000];
    VAR speeddata v57:=[800,500,5000,1000];
    VAR speeddata v58:=[4,500,5000,1000];
    VAR speeddata v59:=[4,500,5000,1000];
    VAR speeddata v60:=[800,500,5000,1000];
    VAR speeddata v61:=[800,500,5000,1000];
    VAR speeddata v62:=[800,500,5000,1000];
    VAR speeddata v63:=[800,500,5000,1000];
    VAR speeddata v64:=[800,500,5000,1000];
    VAR speeddata v65:=[4,500,5000,1000];
    VAR speeddata v66:=[4,500,5000,1000];
    VAR speeddata v67:=[800,500,5000,1000];
    VAR speeddata v68:=[800,500,5000,1000];
    VAR speeddata v69:=[800,500,5000,1000];
    VAR speeddata v70:=[800,500,5000,1000];
    VAR speeddata v71:=[800,500,5000,1000];
    VAR speeddata v72:=[4,500,5000,1000];
    VAR speeddata v73:=[4,500,5000,1000];
    VAR speeddata v74:=[800,500,5000,1000];
    VAR speeddata v75:=[800,500,5000,1000];
    VAR speeddata v76:=[800,500,5000,1000];
    VAR speeddata v77:=[800,500,5000,1000];
    VAR speeddata v78:=[800,500,5000,1000];
    VAR speeddata v79:=[4,500,5000,1000];
    VAR speeddata v80:=[4,500,5000,1000];
    VAR speeddata v81:=[800,500,5000,1000];
    VAR speeddata v82:=[800,500,5000,1000];
    VAR speeddata v83:=[800,500,5000,1000];
    VAR speeddata v84:=[800,500,5000,1000];
    VAR speeddata v85:=[800,500,5000,1000];
    VAR speeddata v86:=[4,500,5000,1000];
    VAR speeddata v87:=[4,500,5000,1000];
    VAR speeddata v88:=[800,500,5000,1000];
    VAR speeddata v89:=[800,500,5000,1000];
    VAR speeddata v90:=[800,500,5000,1000];
    VAR speeddata v91:=[800,500,5000,1000];
    VAR speeddata v92:=[800,500,5000,1000];
    VAR speeddata v93:=[4,500,5000,1000];
    VAR speeddata v94:=[4,500,5000,1000];
    VAR speeddata v95:=[800,500,5000,1000];
    VAR speeddata v96:=[800,500,5000,1000];
    VAR speeddata v97:=[800,500,5000,1000];
    VAR speeddata v98:=[800,500,5000,1000];
    VAR speeddata v99:=[800,500,5000,1000];
    VAR speeddata v100:=[4,500,5000,1000];
    VAR speeddata v101:=[4,500,5000,1000];
    VAR speeddata v102:=[800,500,5000,1000];
    VAR speeddata v103:=[800,500,5000,1000];
    VAR speeddata v104:=[800,500,5000,1000];
    VAR speeddata v105:=[800,500,5000,1000];
    VAR speeddata v106:=[800,500,5000,1000];
    VAR speeddata v107:=[4,500,5000,1000];
    VAR speeddata v108:=[4,500,5000,1000];
    VAR speeddata v109:=[800,500,5000,1000];
    VAR speeddata v110:=[800,500,5000,1000];
    VAR speeddata v111:=[800,500,5000,1000];
    VAR speeddata v112:=[800,500,5000,1000];
    VAR speeddata v113:=[800,500,5000,1000];
    VAR speeddata v114:=[4,500,5000,1000];
    VAR speeddata v115:=[4,500,5000,1000];
    VAR speeddata v116:=[800,500,5000,1000];
    VAR speeddata v117:=[800,500,5000,1000];
    VAR speeddata v118:=[800,500,5000,1000];
    VAR speeddata v119:=[800,500,5000,1000];
    VAR speeddata v120:=[800,500,5000,1000];
    VAR speeddata v121:=[4,500,5000,1000];
    VAR speeddata v122:=[4,500,5000,1000];
    VAR speeddata v123:=[800,500,5000,1000];
    VAR speeddata v124:=[800,500,5000,1000];
    VAR speeddata v125:=[800,500,5000,1000];
    VAR speeddata v126:=[800,500,5000,1000];
    VAR speeddata v127:=[800,500,5000,1000];
    VAR speeddata v128:=[4,500,5000,1000];
    VAR speeddata v129:=[4,500,5000,1000];
    VAR speeddata v130:=[800,500,5000,1000];
    VAR speeddata v131:=[800,500,5000,1000];
    VAR speeddata v132:=[800,500,5000,1000];
    VAR speeddata v133:=[800,500,5000,1000];
    VAR speeddata v134:=[800,500,5000,1000];
    VAR speeddata v135:=[4,500,5000,1000];
    VAR speeddata v136:=[4,500,5000,1000];
    VAR speeddata v137:=[800,500,5000,1000];
    VAR speeddata v138:=[800,500,5000,1000];
    VAR speeddata v139:=[800,500,5000,1000];
ENDMODULE

--- Backups/Rob1/RAPID/TASK1/SYSMOD/StandardJointMoves.sys ---
MODULE StandardJointMoves(SYSMODULE)
    !Home Joint Target
    CONST jointtarget jHome:=[[0,0,0,0,0,0],[9E+09,9E+09,9E+09,9E+09,9E+09,9E+09]];
    !Entry/Exit Joint Targets
    CONST jointtarget jee:=[[-90,14,18,4,-38,0],[9E+09,9E+09,9E+09,9E+09,9E+09,9E+09]];
ENDMODULE

--- Backups/Rob1/RAPID/TASK1/SYSMOD/Tools.sys ---
MODULE Tools(SYSMODULE)
    PERS tooldata MyTool:=[TRUE,[[31.792631019,0,229.638935148],[0.945518576,0,0.325568154,0]],[1,[0,0,1],[1,0,0,0],0,0,0]];
	PERS tooldata PendEff_point:=[TRUE,[[67.056,0,55.372],[0.707106781,0,0.707106781,0]],[1,[0,0,1],[1,0,0,0],0,0,0]];
	PERS tooldata ExternalFedTool:=[TRUE,[[0,0,0],[1,0,0,0]],[0.001,[0,0,0.001],[1,0,0,0],0,0,0]];
	PERS tooldata DrillTool:=[TRUE,[[67.056,0,55.372],[0.7071,0,0.7071,0]],[1,[0,0,1],[1,0,0,0],0,0,0]];
	PERS wobjdata ExternalFedWobjData:=[FALSE,TRUE,"",[[0,0,0],[1,0,0,0]],[[0,0,0],[1,0,0,0]]];
ENDMODULE

--- Backups/Rob1/RAPID/TASK1/SYSMOD/WorkObjs.sys ---
MODULE WorkObjs(SYSMODULE)
    TASK PERS wobjdata A:=[FALSE,TRUE,"",[[246.014,-596.5,290.101],[0,0,0,1]],[[0,0,0],[1,0,0,0]]];
ENDMODULE

--- Backups/Rob2/RAPID/TASK1/PROGMOD/KyleTargets.mod ---
MODULE KyleTargets

	!Workplan Variables
	CONST string workplanName := "Kyle";
	CONST string workplanUUID := "2871e0b1-ddca-400c-8161-6cdc17f12893";

	!Workingsteps
	CONST string WorkPlan{20,6} := [
		["1","7", "Drilling.8", "84ee9563-7912-44c0-bfcd-293f92d8b13d", "Hole.126", "e36ab6dd-4c22-45de-bb9a-479c95405714"],
		["8","14", "Drilling.13", "7ccdfa8a-1cd0-4d02-a500-c80e233b9fd7", "Hole.131", "c4be57f8-fa2c-406f-958b-f31cab34a103"],
		["15","21", "Drilling.14", "8aaf65a2-9007-4bac-b3e6-82b54667c4fe", "Hole.130", "454ae504-a6e0-4436-86a5-e3b48f3a6ebd"],
		["22","28", "Drilling.9", "4f888b1b-6ab9-4e86-946e-5ff123a5037a", "Hole.127", "08e93d49-b28c-4bd3-b6c6-d75430b53a2a"],
		["29","35", "Drilling.7", "02130e2a-b3d5-4e34-8f53-cfbcf2ec8645", "Hole.125", "21017ae4-2b73-4540-894a-30ebc29570ea"],
		["36","42", "Drilling.12", "e30b7ca7-ddbc-40f5-8f65-344a992b1e61", "Hole.132", "e66331d3-3fdc-412a-b6b2-0661d9428281"],
		["43","49", "Drilling.10", "b91ee5e9-1632-43a6-bfe1-16c34d1e5e2f", "Hole.128", "c3d88a5e-7e8b-41d5-b2dc-b0479c29b49e"],
		["50","56", "Drilling.11", "7425d9a6-1369-462c-aada-26a7e19600fd", "Hole.133", "91a8736d-f4a7-4689-80ff-5676ef598fa4"],
		["57","63", "Drilling.27", "5ca7da6b-cc79-4d4d-a6a5-65927e745900", "Hole.135", "331ef13e-3ab3-4da9-b4fa-780c17cbb45e"],
		["64","70", "Drilling.28", "0ef1a843-f159-42da-bcb9-5e1b1c1a301e", "Hole.136", "273267bc-da8b-478b-8b4c-85da8157c9a8"],
		["71","77", "Drilling.29", "11479f12-cf2b-427e-bcec-a468864a2f6d", "Hole.137", "ae1b5195-bf51-44f8-b490-b9d022c936f5"],
		["78","84", "Drilling.30", "d8138029-1469-4182-9afa-9758c29db750", "Hole.138", "46c2d2d0-291f-4604-8bcb-81b365ac65aa"],
		["85","91", "Drilling.31", "8ddb58e3-7706-4204-9557-33380402deaa", "Hole.143", "b8cd4e05-5960-47a1-9f38-2d3fecb31d31"],
		["92","98", "Drilling.32", "bd18ceba-683d-43f3-ad41-06c60c238459", "Hole.142", "cb399f51-d989-4a53-8519-adc3953d158c"],
		["99","105", "Drilling.33", "954da869-fb1d-46f5-9e46-6bf9dcadccda", "Hole.141", "469b1018-b1f9-41c1-939c-a7f265401ba7"],
		["106","112", "Drilling.34", "4e46309a-1422-44c1-86ed-d1c3dc44e9d8", "Hole.140", "37a3b727-c3a1-4ace-845d-67909f3448ad"],
		["113","119", "Drilling.47", "e199d4d2-363b-4bee-92cd-6f11fd8dd563", "Hole.145", "cc8e4781-ee8a-461a-a242-06836f687ae1"],
		["120","126", "Drilling.48", "6d043768-99d8-4c13-af46-7da20463ca22", "Hole.146", "f61a0d74-4152-4b6e-94ed-418b5255987a"],
		["127","133", "Drilling.49", "2f8af433-5b96-4376-97a8-7eb59b4bf896", "Hole.147", "685632c0-b3c9-4929-8c2a-40f363535f56"],
		["134","140", "Drilling.50", "8566419f-d7a9-4061-8d1e-a84c15c8dc73", "Hole.148", "12ffa80d-2d25-44ad-b7a8-efb1cabf81b5"]
		];

	!Positions
	CONST robtarget WorkingstepRobtargets{140} := [
		[[288.779069493284,152.045401982975,43.701087144004],[0.007422705894557,0.000477984990411884,-0.997905463626588,0.0642601013985811],[0,0,0,0],[9E+09,9E+09,9E+09,9E+09,9E+09,9E+09]],
		[[288.029622843527,145.529890074137,-6.67377200502937],[0.007422705894557,0.000477984990411884,-0.997905463626588,0.0642601013985811],[0,0,0,0],[9E+09,9E+09,9E+09,9E+09,9E+09,9E+09]],
		[[288.029622843527,145.529890074137,-6.67377200502937],[0.007422705894557,0.000477984990411884,-0.997905463626588,0.0642601013985811],[0,0,0,0],[9E+09,9E+09,9E+09,9E+09,9E+09,9E+09]],
		[[287.561218687428,141.457695131113,-38.1580589731752],[0.007422705894557,0.000477984990411884,-0.997905463626588,0.0642601013985811],[0,0,0,0],[9E+09,9E+09,9E+09,9E+09,9E+09,9E+09]],
		[[287.561218687428,141.457695131113,-38.1580589731752],[0.007422705894557,0.000477984990411884,-0.997905463626588,0.0642601013985811],[0,0,0,0],[9E+09,9E+09,9E+09,9E+09,9E+09,9E+09]],
		[[288.029622843527,145.529890074137,-6.67377200502937],[0.007422705894557,0.000477984990411884,-0.997905463626588,0.0642601013985811],[0,0,0,0],[9E+09,9E+09,9E+09,9E+09,9E+09,9E+09]],
		[[288.779069493284,152.045401982975,43.701087144004],[0.007422705894557,0.000477984990411884,-0.997905463626588,0.0642601013985811],[0,0,0,0],[9E+09,9E+09,9E+09,9E+09,9E+09,9E+09]],
		[[241.208709454143,129.914601473053,47.0306171325024],[0.00711216548716867,0.000386768399255158,-0.998499282658082,0.0542996320759508],[0,0,0,0],[9E+09,9E+09,9E+09,9E+09,9E+09,9E+09]],
		[[240.489331593404,124.405758598223,-3.46468112064122],[0.00711216548716867,0.000386768399255158,-0.998499282658082,0.0542996320759508],[0,0,0,0],[9E+09,9E+09,9E+09,9E+09,9E+09,9E+09]],
		[[240.489331593404,124.405758598223,-3.46468112064122],[0.00711216548716867,0.000386768399255158,-0.998499282658082,0.0542996320759508],[0,0,0,0],[9E+09,9E+09,9E+09,9E+09,9E+09,9E+09]],
		[[240.039720430442,120.962731801455,-35.0242425288559],[0.00711216548716867,0.000386768399255158,-0.998499282658082,0.0542996320759508],[0,0,0,0],[9E+09,9E+09,9E+09,9E+09,9E+09,9E+09]],
		[[240.039720430442,120.962731801455,-35.0242425288559],[0.00711216548716867,0.000386768399255158,-0.998499282658082,0.0542996320759508],[0,0,0,0],[9E+09,9E+09,9E+09,9E+09,9E+09,9E+09]],
		[[240.489331593404,124.405758598223,-3.46468112064122],[0.00711216548716867,0.000386768399255158,-0.998499282658082,0.0542996320759508],[0,0,0,0],[9E+09,9E+09,9E+09,9E+09,9E+09,9E+09]],
		[[241.208709454143,129.914601473053,47.0306171325024],[0.00711216548716867,0.000386768399255158,-0.998499282658082,0.0542996320759508],[0,0,0,0],[9E+09,9E+09,9E+09,9E+09,9E+09,9E+09]],
		[[241.16608088718,78.4773374561232,51.5237669183629],[0.00662098912699226,0.00021710380003204,-0.999440902554252,0.0327719036746759],[0,0,0,0],[9E+09,9E+09,9E+09,9E+09,9E+09,9E+09]],
		[[240.494487366864,75.1494275837429,0.837338971379267],[0.00662098912699226,0.00021710380003204,-0.999440902554252,0.0327719036746759],[0,0,0,0],[9E+09,9E+09,9E+09,9E+09,9E+09,9E+09]],
		[[240.494487366864,75.1494275837429,0.837338971379267],[0.00662098912699226,0.00021710380003204,-0.999440902554252,0.0327719036746759],[0,0,0,0],[9E+09,9E+09,9E+09,9E+09,9E+09,9E+09]],
		[[240.074741416666,73.0694839135052,-30.8416784954856],[0.00662098912699226,0.00021710380003204,-0.999440902554252,0.0327719036746759],[0,0,0,0],[9E+09,9E+09,9E+09,9E+09,9E+09,9E+09]],
		[[240.074741416666,73.0694839135052,-30.8416784954856],[0.00662098912699226,0.00021710380003204,-0.999440902554252,0.0327719036746759],[0,0,0,0],[9E+09,9E+09,9E+09,9E+09,9E+09,9E+09]],
		[[240.494487366864,75.1494275837429,0.837338971379267],[0.00662098912699226,0.00021710380003204,-0.999440902554252,0.0327719036746759],[0,0,0,0],[9E+09,9E+09,9E+09,9E+09,9E+09,9E+09]],
		[[241.16608088718,78.4773374561232,51.5237669183629],[0.00662098912699226,0.00021710380003204,-0.999440902554252,0.0327719036746759],[0,0,0,0],[9E+09,9E+09,9E+09,9E+09,9E+09,9E+09]],
		[[289.915081712141,203.37187194352,35.8970963576192],[0.00829344469822132,0.00071684874899254,-0.99625072742016,0.0861115150122795],[0,0,0,0],[9E+09,9E+09,9E+09,9E+09,9E+09,9E+09]],
		[[289.081898579771,194.655140114566,-14.1425318593251],[0.00829344469822132,0.00071684874899254,-0.99625072742016,0.0861115150122795],[0,0,0,0],[9E+09,9E+09,9E+09,9E+09,9E+09,9E+09]],
		[[289.081898579771,194.655140114566,-14.1425318593251],[0.00829344469822132,0.00071684874899254,-0.99625072742016,0.0861115150122795],[0,0,0,0],[9E+09,9E+09,9E+09,9E+09,9E+09,9E+09]],
		[[288.561159122039,189.207182721469,-45.4172994949153],[0.00829344469822132,0.00071684874899254,-0.99625072742016,0.0861115150122795],[0,0,0,0],[9E+09,9E+09,9E+09,9E+09,9E+09,9E+09]],
		[[288.561159122039,189.207182721469,-45.4172994949153],[0.00829344469822132,0.00071684874899254,-0.99625072742016,0.0861115150122795],[0,0,0,0],[9E+09,9E+09,9E+09,9E+09,9E+09,9E+09]],
		[[289.081898579771,194.655140114566,-14.1425318593251],[0.00829344469822132,0.00071684874899254,-0.99625072742016,0.0861115150122795],[0,0,0,0],[9E+09,9E+09,9E+09,9E+09,9E+09,9E+09]],
		[[289.915081712141,203.37187194352,35.8970963576192],[0.00829344469822132,0.00071684874899254,-0.99625072742016,0.0861115150122795],[0,0,0,0],[9E+09,9E+09,9E+09,9E+09,9E+09,9E+09]],
		[[289.138188356465,99.8323134359238,49.2767143787854],[0.00680464181526441,0.000287089635706398,-0.999088004780398,0.0421517868331755],[0,0,0,0],[9E+09,9E+09,9E+09,9E+09,9E+09,9E+09]],
		[[288.448696753655,95.553399144166,-1.33806107081477],[0.00680464181526441,0.000287089635706398,-0.999088004780398,0.0421517868331755],[0,0,0,0],[9E+09,9E+09,9E+09,9E+09,9E+09,9E+09]],
		[[288.448696753655,95.553399144166,-1.33806107081477],[0.00680464181526441,0.000287089635706398,-0.999088004780398,0.0421517868331755],[0,0,0,0],[9E+09,9E+09,9E+09,9E+09,9E+09,9E+09]],
		[[288.017764501897,92.8790777118172,-32.9722957268149],[0.00680464181526441,0.000287089635706398,-0.999088004780398,0.0421517868331755],[0,0,0,0],[9E+09,9E+09,9E+09,9E+09,9E+09,9E+09]],
		[[288.017764501897,92.8790777118172,-32.9722957268149],[0.00680464181526441,0.000287089635706398,-0.999088004780398,0.0421517868331755],[0,0,0,0],[9E+09,9E+09,9E+09,9E+09,9E+09,9E+09]],
		[[288.448696753655,95.553399144166,-1.33806107081477],[0.00680464181526441,0.000287089635706398,-0.999088004780398,0.0421517868331755],[0,0,0,0],[9E+09,9E+09,9E+09,9E+09,9E+09,9E+09]],
		[[289.138188356465,99.8323134359238,49.2767143787854],[0.00680464181526441,0.000287089635706398,-0.999088004780398,0.0421517868331755],[0,0,0,0],[9E+09,9E+09,9E+09,9E+09,9E+09,9E+09]],
		[[241.289915734788,182.554869058621,40.1026325032385],[0.00787523856525625,0.000603576012444046,-0.997044757638711,0.0764157547806785],[0,0,0,0],[9E+09,9E+09,9E+09,9E+09,9E+09,9E+09]],
		[[240.496842125603,174.813489467987,-10.0977865815075],[0.00787523856525625,0.000603576012444046,-0.997044757638711,0.0764157547806785],[0,0,0,0],[9E+09,9E+09,9E+09,9E+09,9E+09,9E+09]],
		[[240.496842125603,174.813489467987,-10.0977865815075],[0.00787523856525625,0.000603576012444046,-0.997044757638711,0.0764157547806785],[0,0,0,0],[9E+09,9E+09,9E+09,9E+09,9E+09,9E+09]],
		[[240.001171119863,169.975127223841,-41.4730485094737],[0.00787523856525625,0.000603576012444046,-0.997044757638711,0.0764157547806785],[0,0,0,0],[9E+09,9E+09,9E+09,9E+09,9E+09,9E+09]],
		[[240.001171119863,169.975127223841,-41.4730485094737],[0.00787523856525625,0.000603576012444046,-0.997044757638711,0.0764157547806785],[0,0,0,0],[9E+09,9E+09,9E+09,9E+09,9E+09,9E+09]],
		[[240.496842125603,174.813489467987,-10.0977865815075],[0.00787523856525625,0.000603576012444046,-0.997044757638711,0.0764157547806785],[0,0,0,0],[9E+09,9E+09,9E+09,9E+09,9E+09,9E+09]],
		[[241.289915734788,182.554869058621,40.1026325032385],[0.00787523856525625,0.000603576012444046,-0.997044757638711,0.0764157547806785],[0,0,0,0],[9E+09,9E+09,9E+09,9E+09,9E+09,9E+09]],
		[[289.309102101314,245.858135120208,27.7054804314411],[0.00921908733036795,0.000966562056112772,-0.994506082335781,0.104267571103021],[0,0,0,0],[9E+09,9E+09,9E+09,9E+09,9E+09,9E+09]],
		[[288.387828114989,235.321844841818,-21.9813170243381],[0.00921908733036795,0.000966562056112772,-0.994506082335781,0.104267571103021],[0,0,0,0],[9E+09,9E+09,9E+09,9E+09,9E+09,9E+09]],
		[[288.387828114989,235.321844841818,-21.9813170243381],[0.00921908733036795,0.000966562056112772,-0.994506082335781,0.104267571103021],[0,0,0,0],[9E+09,9E+09,9E+09,9E+09,9E+09,9E+09]],
		[[287.812031873535,228.736663417825,-53.0355654342003],[0.00921908733036795,0.000966562056112772,-0.994506082335781,0.104267571103021],[0,0,0,0],[9E+09,9E+09,9E+09,9E+09,9E+09,9E+09]],
		[[287.812031873535,228.736663417825,-53.0355654342003],[0.00921908733036795,0.000966562056112772,-0.994506082335781,0.104267571103021],[0,0,0,0],[9E+09,9E+09,9E+09,9E+09,9E+09,9E+09]],
		[[288.387828114989,235.321844841818,-21.9813170243381],[0.00921908733036795,0.000966562056112772,-0.994506082335781,0.104267571103021],[0,0,0,0],[9E+09,9E+09,9E+09,9E+09,9E+09,9E+09]],
		[[289.309102101314,245.858135120208,27.7054804314411],[0.00921908733036795,0.000966562056112772,-0.994506082335781,0.104267571103021],[0,0,0,0],[9E+09,9E+09,9E+09,9E+09,9E+09,9E+09]],
		[[241.458489628179,256.577531419905,26.2903440426919],[0.0094165728968686,0.00102020140999334,-0.99413767750685,0.107705921402901],[0,0,0,0],[9E+09,9E+09,9E+09,9E+09,9E+09,9E+09]],
		[[240.518538429408,245.697784689916,-23.3220294425105],[0.0094165728968686,0.00102020140999334,-0.99413767750685,0.107705921402901],[0,0,0,0],[9E+09,9E+09,9E+09,9E+09,9E+09,9E+09]],
		[[240.518538429408,245.697784689916,-23.3220294425105],[0.0094165728968686,0.00102020140999334,-0.99413767750685,0.107705921402901],[0,0,0,0],[9E+09,9E+09,9E+09,9E+09,9E+09,9E+09]],
		[[239.931068930175,238.897942983672,-54.3297628707619],[0.0094165728968686,0.00102020140999334,-0.99413767750685,0.107705921402901],[0,0,0,0],[9E+09,9E+09,9E+09,9E+09,9E+09,9E+09]],
		[[239.931068930175,238.897942983672,-54.3297628707619],[0.0094165728968686,0.00102020140999334,-0.99413767750685,0.107705921402901],[0,0,0,0],[9E+09,9E+09,9E+09,9E+09,9E+09,9E+09]],
		[[240.518538429408,245.697784689916,-23.3220294425105],[0.0094165728968686,0.00102020140999334,-0.99413767750685,0.107705921402901],[0,0,0,0],[9E+09,9E+09,9E+09,9E+09,9E+09,9E+09]],
		[[241.458489628179,256.577531419905,26.2903440426919],[0.0094165728968686,0.00102020140999334,-0.99413767750685,0.107705921402901],[0,0,0,0],[9E+09,9E+09,9E+09,9E+09,9E+09,9E+09]],
		[[385.659328209428,81.9362218762582,49.3667840745575],[0.00666644321018516,0.000235774252738867,-0.999352927467223,0.0353444381497125],[0,0,0,0],[9E+09,9E+09,9E+09,9E+09,9E+09,9E+09]],
		[[384.983302512521,78.3473909020153,-1.30177897488602],[0.00666644321018516,0.000235774252738867,-0.999352927467223,0.0353444381497125],[0,0,0,0],[9E+09,9E+09,9E+09,9E+09,9E+09,9E+09]],
		[[384.983302512521,78.3473909020153,-1.30177897488602],[0.00666644321018516,0.000235774252738867,-0.999352927467223,0.0353444381497125],[0,0,0,0],[9E+09,9E+09,9E+09,9E+09,9E+09,9E+09]],
		[[384.560786451954,76.1043715431133,-32.9696308807882],[0.00666644321018516,0.000235774252738867,-0.999352927467223,0.0353444381497125],[0,0,0,0],[9E+09,9E+09,9E+09,9E+09,9E+09,9E+09]],
		[[384.560786451954,76.1043715431133,-32.9696308807882],[0.00666644321018516,0.000235774252738867,-0.999352927467223,0.0353444381497125],[0,0,0,0],[9E+09,9E+09,9E+09,9E+09,9E+09,9E+09]],
		[[384.983302512521,78.3473909020153,-1.30177897488602],[0.00666644321018516,0.000235774252738867,-0.999352927467223,0.0353444381497125],[0,0,0,0],[9E+09,9E+09,9E+09,9E+09,9E+09,9E+09]],
		[[385.659328209428,81.9362218762582,49.3667840745575],[0.00666644321018516,0.000235774252738867,-0.999352927467223,0.0353444381497125],[0,0,0,0],[9E+09,9E+09,9E+09,9E+09,9E+09,9E+09]],
		[[385.705942714164,121.3363389992,45.8993369958386],[0.00705746724934637,0.000370148416132423,-0.998602508304339,0.0523744742642432],[0,0,0,0],[9E+09,9E+09,9E+09,9E+09,9E+09,9E+09]],
		[[384.991875748216,116.022263401137,-4.61690503488058],[0.00705746724934637,0.000370148416132423,-0.998602508304339,0.0523744742642432],[0,0,0,0],[9E+09,9E+09,9E+09,9E+09,9E+09,9E+09]],
		[[384.991875748216,116.022263401137,-4.61690503488058],[0.00705746724934637,0.000370148416132423,-0.998602508304339,0.0523744742642432],[0,0,0,0],[9E+09,9E+09,9E+09,9E+09,9E+09,9E+09]],
		[[384.545583894497,112.700966152347,-36.1895563040799],[0.00705746724934637,0.000370148416132423,-0.998602508304339,0.0523744742642432],[0,0,0,0],[9E+09,9E+09,9E+09,9E+09,9E+09,9E+09]],
		[[384.545583894497,112.700966152347,-36.1895563040799],[0.00705746724934637,0.000370148416132423,-0.998602508304339,0.0523744742642432],[0,0,0,0],[9E+09,9E+09,9E+09,9E+09,9E+09,9E+09]],
		[[384.991875748216,116.022263401137,-4.61690503488058],[0.00705746724934637,0.000370148416132423,-0.998602508304339,0.0523744742642432],[0,0,0,0],[9E+09,9E+09,9E+09,9E+09,9E+09,9E+09]],
		[[385.705942714164,121.3363389992,45.8993369958386],[0.00705746724934637,0.000370148416132423,-0.998602508304339,0.0523744742642432],[0,0,0,0],[9E+09,9E+09,9E+09,9E+09,9E+09,9E+09]],
		[[385.786606171087,170.92295449455,39.5986687515689],[0.0077728569445215,0.000575867762347651,-0.997236511782182,0.073882275545262],[0,0,0,0],[9E+09,9E+09,9E+09,9E+09,9E+09,9E+09]],
		[[385.003389010044,163.436804479832,-10.6406000412369],[0.0077728569445215,0.000575867762347651,-0.997236511782182,0.073882275545262],[0,0,0,0],[9E+09,9E+09,9E+09,9E+09,9E+09,9E+09]],
		[[385.003389010044,163.436804479832,-10.6406000412369],[0.0077728569445215,0.000575867762347651,-0.997236511782182,0.073882275545262],[0,0,0,0],[9E+09,9E+09,9E+09,9E+09,9E+09,9E+09]],
		[[384.513878284388,158.757960720632,-42.0401430367406],[0.0077728569445215,0.000575867762347651,-0.997236511782182,0.073882275545262],[0,0,0,0],[9E+09,9E+09,9E+09,9E+09,9E+09,9E+09]],
		[[384.513878284388,158.757960720632,-42.0401430367406],[0.0077728569445215,0.000575867762347651,-0.997236511782182,0.073882275545262],[0,0,0,0],[9E+09,9E+09,9E+09,9E+09,9E+09,9E+09]],
		[[385.003389010044,163.436804479832,-10.6406000412369],[0.0077728569445215,0.000575867762347651,-0.997236511782182,0.073882275545262],[0,0,0,0],[9E+09,9E+09,9E+09,9E+09,9E+09,9E+09]],
		[[385.786606171087,170.92295449455,39.5986687515689],[0.0077728569445215,0.000575867762347651,-0.997236511782182,0.073882275545262],[0,0,0,0],[9E+09,9E+09,9E+09,9E+09,9E+09,9E+09]],
		[[377.811662051271,247.005082716161,25.8049759829888],[0.00936607002242295,0.00100689956012748,-0.994226831681083,0.106884377020243],[0,0,0,0],[9E+09,9E+09,9E+09,9E+09,9E+09,9E+09]],
		[[376.876497420054,236.207365300938,-23.8254054958343],[0.00936607002242295,0.00100689956012748,-0.994226831681083,0.106884377020243],[0,0,0,0],[9E+09,9E+09,9E+09,9E+09,9E+09,9E+09]],
		[[376.876497420054,236.207365300938,-23.8254054958343],[0.00936607002242295,0.00100689956012748,-0.994226831681083,0.106884377020243],[0,0,0,0],[9E+09,9E+09,9E+09,9E+09,9E+09,9E+09]],
		[[376.292019525545,229.458791916423,-54.8443939200984],[0.00936607002242295,0.00100689956012748,-0.994226831681083,0.106884377020243],[0,0,0,0],[9E+09,9E+09,9E+09,9E+09,9E+09,9E+09]],
		[[376.292019525545,229.458791916423,-54.8443939200984],[0.00936607002242295,0.00100689956012748,-0.994226831681083,0.106884377020243],[0,0,0,0],[9E+09,9E+09,9E+09,9E+09,9E+09,9E+09]],
		[[376.876497420054,236.207365300938,-23.8254054958343],[0.00936607002242295,0.00100689956012748,-0.994226831681083,0.106884377020243],[0,0,0,0],[9E+09,9E+09,9E+09,9E+09,9E+09,9E+09]],
		[[377.811662051271,247.005082716161,25.8049759829888],[0.00936607002242295,0.00100689956012748,-0.994226831681083,0.106884377020243],[0,0,0,0],[9E+09,9E+09,9E+09,9E+09,9E+09,9E+09]],
		[[480.170049765267,240.852707828735,25.2149600674652],[0.00935279474907906,0.00100366331647834,-0.99424737884142,0.106694271436163],[0,0,0,0],[9E+09,9E+09,9E+09,9E+09,9E+09,9E+09]],
		[[479.236152061027,230.073975332924,-24.4195718721205],[0.00935279474907906,0.00100366331647834,-0.99424737884142,0.106694271436163],[0,0,0,0],[9E+09,9E+09,9E+09,9E+09,9E+09,9E+09]],
		[[479.236152061027,230.073975332924,-24.4195718721205],[0.00935279474907906,0.00100366331647834,-0.99424737884142,0.106694271436163],[0,0,0,0],[9E+09,9E+09,9E+09,9E+09,9E+09,9E+09]],
		[[478.652465995876,223.337267523042,-55.4411543343616],[0.00935279474907906,0.00100366331647834,-0.99424737884142,0.106694271436163],[0,0,0,0],[9E+09,9E+09,9E+09,9E+09,9E+09,9E+09]],
		[[478.652465995876,223.337267523042,-55.4411543343616],[0.00935279474907906,0.00100366331647834,-0.99424737884142,0.106694271436163],[0,0,0,0],[9E+09,9E+09,9E+09,9E+09,9E+09,9E+09]],
		[[479.236152061027,230.073975332924,-24.4195718721205],[0.00935279474907906,0.00100366331647834,-0.99424737884142,0.106694271436163],[0,0,0,0],[9E+09,9E+09,9E+09,9E+09,9E+09,9E+09]],
		[[480.170049765267,240.852707828735,25.2149600674652],[0.00935279474907906,0.00100366331647834,-0.99424737884142,0.106694271436163],[0,0,0,0],[9E+09,9E+09,9E+09,9E+09,9E+09,9E+09]],
		[[480.004815039626,167.740024424446,38.6041144078019],[0.00778003061909403,0.000578044083313996,-0.99722089826046,0.0740919500432094],[0,0,0,0],[9E+09,9E+09,9E+09,9E+09,9E+09,9E+09]],
		[[479.220912039579,160.232745745701,-11.6319907649338],[0.00778003061909403,0.000578044083313996,-0.99722089826046,0.0740919500432094],[0,0,0,0],[9E+09,9E+09,9E+09,9E+09,9E+09,9E+09]],
		[[479.220912039579,160.232745745701,-11.6319907649338],[0.00778003061909403,0.000578044083313996,-0.99722089826046,0.0740919500432094],[0,0,0,0],[9E+09,9E+09,9E+09,9E+09,9E+09,9E+09]],
		[[478.73097266455,155.540696571485,-43.0295564978937],[0.00778003061909403,0.000578044083313996,-0.99722089826046,0.0740919500432094],[0,0,0,0],[9E+09,9E+09,9E+09,9E+09,9E+09,9E+09]],
		[[478.73097266455,155.540696571485,-43.0295564978937],[0.00778003061909403,0.000578044083313996,-0.99722089826046,0.0740919500432094],[0,0,0,0],[9E+09,9E+09,9E+09,9E+09,9E+09,9E+09]],
		[[479.220912039579,160.232745745701,-11.6319907649338],[0.00778003061909403,0.000578044083313996,-0.99722089826046,0.0740919500432094],[0,0,0,0],[9E+09,9E+09,9E+09,9E+09,9E+09,9E+09]],
		[[480.004815039626,167.740024424446,38.6041144078019],[0.00778003061909403,0.000578044083313996,-0.99722089826046,0.0740919500432094],[0,0,0,0],[9E+09,9E+09,9E+09,9E+09,9E+09,9E+09]],
		[[479.919259856698,121.968377201349,44.4964931486716],[0.00709667369513751,0.000382372295419974,-0.998526380753501,0.0538010962082301],[0,0,0,0],[9E+09,9E+09,9E+09,9E+09,9E+09,9E+09]],
		[[479.201390441381,116.509965212552,-6.00430290508506],[0.00709667369513751,0.000382372295419974,-0.998526380753501,0.0538010962082301],[0,0,0,0],[9E+09,9E+09,9E+09,9E+09,9E+09,9E+09]],
		[[479.201390441381,116.509965212552,-6.00430290508506],[0.00709667369513751,0.000382372295419974,-0.998526380753501,0.0538010962082301],[0,0,0,0],[9E+09,9E+09,9E+09,9E+09,9E+09,9E+09]],
		[[478.752722056809,113.098457719554,-37.5673004386829],[0.00709667369513751,0.000382372295419974,-0.998526380753501,0.0538010962082301],[0,0,0,0],[9E+09,9E+09,9E+09,9E+09,9E+09,9E+09]],
		[[478.752722056809,113.098457719554,-37.5673004386829],[0.00709667369513751,0.000382372295419974,-0.998526380753501,0.0538010962082301],[0,0,0,0],[9E+09,9E+09,9E+09,9E+09,9E+09,9E+09]],
		[[479.201390441381,116.509965212552,-6.00430290508506],[0.00709667369513751,0.000382372295419974,-0.998526380753501,0.0538010962082301],[0,0,0,0],[9E+09,9E+09,9E+09,9E+09,9E+09,9E+09]],
		[[479.919259856698,121.968377201349,44.4964931486716],[0.00709667369513751,0.000382372295419974,-0.998526380753501,0.0538010962082301],[0,0,0,0],[9E+09,9E+09,9E+09,9E+09,9E+09,9E+09]],
		[[479.875986083091,82.7441856052948,48.0496180783819],[0.00668739513582172,0.000244089648411723,-0.999312165570881,0.0364748530987777],[0,0,0,0],[9E+09,9E+09,9E+09,9E+09,9E+09,9E+09]],
		[[479.197918637486,79.0407236941793,-2.6106680875305],[0.00668739513582172,0.000244089648411723,-0.999312165570881,0.0364748530987777],[0,0,0,0],[9E+09,9E+09,9E+09,9E+09,9E+09,9E+09]],
		[[479.197918637486,79.0407236941793,-2.6106680875305],[0.00668739513582172,0.000244089648411723,-0.999312165570881,0.0364748530987777],[0,0,0,0],[9E+09,9E+09,9E+09,9E+09,9E+09,9E+09]],
		[[478.774126483985,76.7260599997321,-34.2733469412257],[0.00668739513582172,0.000244089648411723,-0.999312165570881,0.0364748530987777],[0,0,0,0],[9E+09,9E+09,9E+09,9E+09,9E+09,9E+09]],
		[[478.774126483985,76.7260599997321,-34.2733469412257],[0.00668739513582172,0.000244089648411723,-0.999312165570881,0.0364748530987777],[0,0,0,0],[9E+09,9E+09,9E+09,9E+09,9E+09,9E+09]],
		[[479.197918637486,79.0407236941793,-2.6106680875305],[0.00668739513582172,0.000244089648411723,-0.999312165570881,0.0364748530987777],[0,0,0,0],[9E+09,9E+09,9E+09,9E+09,9E+09,9E+09]],
		[[479.875986083091,82.7441856052948,48.0496180783819],[0.00668739513582172,0.000244089648411723,-0.999312165570881,0.0364748530987777],[0,0,0,0],[9E+09,9E+09,9E+09,9E+09,9E+09,9E+09]],
		[[586.795866652297,78.1720086574168,46.9499170079332],[0.00666571377515568,0.000235671494483464,-0.99935333985005,0.0353329145325675],[0,0,0,0],[9E+09,9E+09,9E+09,9E+09,9E+09,9E+09]],
		[[586.119914093827,74.5843463317669,-3.71872977857378],[0.00666571377515568,0.000235671494483464,-0.99935333985005,0.0353329145325675],[0,0,0,0],[9E+09,9E+09,9E+09,9E+09,9E+09,9E+09]],
		[[586.119914093827,74.5843463317669,-3.71872977857378],[0.00666571377515568,0.000235671494483464,-0.99935333985005,0.0353329145325675],[0,0,0,0],[9E+09,9E+09,9E+09,9E+09,9E+09,9E+09]],
		[[585.697443744781,72.3420573782357,-35.3866340201408],[0.00666571377515568,0.000235671494483464,-0.99935333985005,0.0353329145325675],[0,0,0,0],[9E+09,9E+09,9E+09,9E+09,9E+09,9E+09]],
		[[585.697443744781,72.3420573782357,-35.3866340201408],[0.00666571377515568,0.000235671494483464,-0.99935333985005,0.0353329145325675],[0,0,0,0],[9E+09,9E+09,9E+09,9E+09,9E+09,9E+09]],
		[[586.119914093827,74.5843463317669,-3.71872977857378],[0.00666571377515568,0.000235671494483464,-0.99935333985005,0.0353329145325675],[0,0,0,0],[9E+09,9E+09,9E+09,9E+09,9E+09,9E+09]],
		[[586.795866652297,78.1720086574168,46.9499170079332],[0.00666571377515568,0.000235671494483464,-0.99935333985005,0.0353329145325675],[0,0,0,0],[9E+09,9E+09,9E+09,9E+09,9E+09,9E+09]],
		[[582.277502827268,118.969427450682,43.3656713654528],[0.00709470104640348,0.0003819253989814,-0.99852896922153,0.0537532973448111],[0,0,0,0],[9E+09,9E+09,9E+09,9E+09,9E+09,9E+09]],
		[[581.559827374303,113.515850932253,-7.13564985589618],[0.00709470104640348,0.0003819253989814,-0.99852896922153,0.0537532973448111],[0,0,0,0],[9E+09,9E+09,9E+09,9E+09,9E+09,9E+09]],
		[[581.559827374303,113.515850932253,-7.13564985589618],[0.00709470104640348,0.0003819253989814,-0.99852896922153,0.0537532973448111],[0,0,0,0],[9E+09,9E+09,9E+09,9E+09,9E+09,9E+09]],
		[[581.1112802162,110.107365608236,-38.6989756192391],[0.00709470104640348,0.0003819253989814,-0.99852896922153,0.0537532973448111],[0,0,0,0],[9E+09,9E+09,9E+09,9E+09,9E+09,9E+09]],
		[[581.1112802162,110.107365608236,-38.6989756192391],[0.00709470104640348,0.0003819253989814,-0.99852896922153,0.0537532973448111],[0,0,0,0],[9E+09,9E+09,9E+09,9E+09,9E+09,9E+09]],
		[[581.559827374303,113.515850932253,-7.13564985589618],[0.00709470104640348,0.0003819253989814,-0.99852896922153,0.0537532973448111],[0,0,0,0],[9E+09,9E+09,9E+09,9E+09,9E+09,9E+09]],
		[[582.277502827268,118.969427450682,43.3656713654528],[0.00709470104640348,0.0003819253989814,-0.99852896922153,0.0537532973448111],[0,0,0,0],[9E+09,9E+09,9E+09,9E+09,9E+09,9E+09]],
		[[586.927237975716,164.1291021749,37.4752655648295],[0.00778853013651704,0.000580626521977126,-0.997202342888956,0.0743403592130852],[0,0,0,0],[9E+09,9E+09,9E+09,9E+09,9E+09,9E+09]],
		[[586.142522601734,156.596792870165,-12.7570799738735],[0.00778853013651704,0.000580626521977126,-0.997202342888956,0.0743403592130852],[0,0,0,0],[9E+09,9E+09,9E+09,9E+09,9E+09,9E+09]],
		[[586.142522601734,156.596792870165,-12.7570799738735],[0.00778853013651704,0.000580626521977126,-0.997202342888956,0.0743403592130852],[0,0,0,0],[9E+09,9E+09,9E+09,9E+09,9E+09,9E+09]],
		[[585.652075492993,151.889099554705,-44.1522959355627],[0.00778853013651704,0.000580626521977126,-0.997202342888956,0.0743403592130852],[0,0,0,0],[9E+09,9E+09,9E+09,9E+09,9E+09,9E+09]],
		[[585.652075492993,151.889099554705,-44.1522959355627],[0.00778853013651704,0.000580626521977126,-0.997202342888956,0.0743403592130852],[0,0,0,0],[9E+09,9E+09,9E+09,9E+09,9E+09,9E+09]],
		[[586.142522601734,156.596792870165,-12.7570799738735],[0.00778853013651704,0.000580626521977126,-0.997202342888956,0.0743403592130852],[0,0,0,0],[9E+09,9E+09,9E+09,9E+09,9E+09,9E+09]],
		[[586.927237975716,164.1291021749,37.4752655648295],[0.00778853013651704,0.000580626521977126,-0.997202342888956,0.0743403592130852],[0,0,0,0],[9E+09,9E+09,9E+09,9E+09,9E+09,9E+09]],
		[[590.794286307596,244.05726888917,22.3952123523095],[0.00960319833789452,0.00107271202908935,-0.993772536259963,0.111007990910686],[0,0,0,0],[9E+09,9E+09,9E+09,9E+09,9E+09,9E+09]],
		[[589.83677588721,232.848046284667,-27.1434241085131],[0.00960319833789452,0.00107271202908935,-0.993772536259963,0.111007990910686],[0,0,0,0],[9E+09,9E+09,9E+09,9E+09,9E+09,9E+09]],
		[[589.83677588721,232.848046284667,-27.1434241085131],[0.00960319833789452,0.00107271202908935,-0.993772536259963,0.111007990910686],[0,0,0,0],[9E+09,9E+09,9E+09,9E+09,9E+09,9E+09]],
		[[589.238331874469,225.842282156853,-58.105071896527],[0.00960319833789452,0.00107271202908935,-0.993772536259963,0.111007990910686],[0,0,0,0],[9E+09,9E+09,9E+09,9E+09,9E+09,9E+09]],
		[[589.238331874469,225.842282156853,-58.105071896527],[0.00960319833789452,0.00107271202908935,-0.993772536259963,0.111007990910686],[0,0,0,0],[9E+09,9E+09,9E+09,9E+09,9E+09,9E+09]],
		[[589.83677588721,232.848046284667,-27.1434241085131],[0.00960319833789452,0.00107271202908935,-0.993772536259963,0.111007990910686],[0,0,0,0],[9E+09,9E+09,9E+09,9E+09,9E+09,9E+09]],
		[[590.794286307596,244.05726888917,22.3952123523095],[0.00960319833789452,0.00107271202908935,-0.993772536259963,0.111007990910686],[0,0,0,0],[9E+09,9E+09,9E+09,9E+09,9E+09,9E+09]]
		];

